LIN {X 0,Y 523.259,Z 482.213,A -85,B 0,C 180,E1 -4769.999,E2 -4769.999} C_VEL
LIN {X 0,Y 523.274,Z 481.391,A -85,B 0,C 180,E1 -4771.538,E2 -4771.538} C_VEL
LIN {X 0,Y 523.335,Z 480.397,A -85,B 0,C 180,E1 -4772.307,E2 -4772.307} C_VEL
LIN {X 0,Y 523.367,Z 478.999,A -85,B 0,C 180,E1 -4773.077,E2 -4773.077} C_VEL
LIN {X 0,Y 523.423,Z 476.057,A -85,B 0,C 180,E1 -4774.233,E2 -4774.233} C_VEL
LIN {X 0,Y 523.455,Z 472.072,A -85,B 0,C 180,E1 -4775.391,E2 -4775.391} C_VEL
LIN {X 0,Y 523.508,Z 466.867,A -85,B 0,C 180,E1 -4776.566,E2 -4776.566} C_VEL
LIN {X 0,Y 523.611,Z 460.488,A -85,B 0,C 180,E1 -4777.711,E2 -4777.711} C_VEL
LIN {X 0,Y 523.8,Z 452.437,A -85,B 0,C 180,E1 -4778.874,E2 -4778.874} C_VEL
LIN {X 0,Y 523.986,Z 444.235,A -85,B 0,C 180,E1 -4779.844,E2 -4779.844} C_VEL
LIN {X 0,Y 524.294,Z 434.24,A -85,B 0,C 180,E1 -4780.814,E2 -4780.814} C_VEL
LIN {X 0,Y 524.558,Z 422.98,A -85,B 0,C 180,E1 -4781.687,E2 -4781.687} C_VEL
LIN {X 0,Y 524.835,Z 411.905,A -85,B 0,C 180,E1 -4782.369,E2 -4782.369} C_VEL
LIN {X 0,Y 525.111,Z 399.665,A -85,B 0,C 180,E1 -4782.952,E2 -4782.952} C_VEL
LIN {X 0,Y 525.344,Z 387.753,A -85,B 0,C 180,E1 -4783.364,E2 -4783.364} C_VEL
LIN {X 0,Y 525.517,Z 374.759,A -85,B 0,C 180,E1 -4783.655,E2 -4783.655} C_VEL
LIN {X 0,Y 525.809,Z 279.444,A -85,B 0,C 180,E1 -4784.972,E2 -4784.972} C_VEL
LIN {X 0,Y 524.262,Z 268.901,A -85,B 0,C 180,E1 -4785.178,E2 -4785.178} C_VEL
LIN {X 0,Y 524.642,Z 248.982,A -85,B 0,C 180,E1 -4788.123,E2 -4788.123} C_VEL
LIN {X 0,Y 525.091,Z 228.582,A -85,B 0,C 180,E1 -4791.181,E2 -4791.181} C_VEL
LIN {X 0,Y 525.423,Z 212.316,A -85,B 0,C 180,E1 -4793.654,E2 -4793.654} C_VEL
LIN {X 0,Y 523.985,Z 204.216,A -85,B 0,C 180,E1 -4794.988,E2 -4794.988} C_VEL
LIN {X 0,Y 523.955,Z 204.222,A -85,B 0,C 180,E1 -4797.995,E2 -4797.995} C_VEL
LIN {X 0,Y 523.926,Z 204.218,A -85,B 0,C 180,E1 -4800.851,E2 -4800.851} C_VEL
LIN {X 0,Y 523.942,Z 204.22,A -85,B 0,C 180,E1 -4803.731,E2 -4803.731} C_VEL
LIN {X 0,Y 523.898,Z 204.224,A -85,B 0,C 180,E1 -4806.4,E2 -4806.4} C_VEL
LIN {X 0,Y 523.896,Z 204.221,A -85,B 0,C 180,E1 -4809.08,E2 -4809.08} C_VEL
LIN {X 0,Y 523.926,Z 204.223,A -85,B 0,C 180,E1 -4812.114,E2 -4812.114} C_VEL
LIN {X 0,Y 523.922,Z 204.22,A -85,B 0,C 180,E1 -4815.305,E2 -4815.305} C_VEL
LIN {X 0,Y 523.946,Z 204.215,A -85,B 0,C 180,E1 -4818.682,E2 -4818.682} C_VEL
LIN {X 0,Y 523.916,Z 204.22,A -85,B 0,C 180,E1 -4821.072,E2 -4821.072} C_VEL
LIN {X 0,Y 523.887,Z 204.229,A -85,B 0,C 180,E1 -4823.824,E2 -4823.824} C_VEL
LIN {X 0,Y 523.904,Z 204.22,A -85,B 0,C 180,E1 -4826.633,E2 -4826.633} C_VEL
LIN {X 0,Y 523.918,Z 204.224,A -85,B 0,C 180,E1 -4829.353,E2 -4829.353} C_VEL
LIN {X 0,Y 523.932,Z 204.217,A -85,B 0,C 180,E1 -4832.277,E2 -4832.277} C_VEL
LIN {X 0,Y 523.904,Z 204.22,A -85,B 0,C 180,E1 -4834.579,E2 -4834.579} C_VEL
LIN {X 0,Y 523.913,Z 204.223,A -85,B 0,C 180,E1 -4837.107,E2 -4837.107} C_VEL
LIN {X 0,Y 523.925,Z 204.22,A -85,B 0,C 180,E1 -4839.863,E2 -4839.863} C_VEL
LIN {X 0,Y 523.941,Z 204.218,A -85,B 0,C 180,E1 -4842.836,E2 -4842.836} C_VEL
LIN {X 0,Y 523.945,Z 204.223,A -85,B 0,C 180,E1 -4845.235,E2 -4845.235} C_VEL
LIN {X 0,Y 523.959,Z 204.213,A -85,B 0,C 180,E1 -4848.393,E2 -4848.393} C_VEL
LIN {X 0,Y 523.95,Z 204.219,A -85,B 0,C 180,E1 -4851.515,E2 -4851.515} C_VEL
LIN {X 0,Y 523.993,Z 204.21,A -85,B 0,C 180,E1 -4853.84,E2 -4853.84} C_VEL
LIN {X 0,Y 524.021,Z 204.212,A -85,B 0,C 180,E1 -4856.925,E2 -4856.925} C_VEL
LIN {X 0,Y 524.047,Z 204.202,A -85,B 0,C 180,E1 -4860,E2 -4860} C_VEL
LIN {X 0,Y 524.019,Z 204.214,A -85,B 0,C 180,E1 -4863.075,E2 -4863.075} C_VEL
LIN {X 0,Y 523.985,Z 204.21,A -85,B 0,C 180,E1 -4866.16,E2 -4866.16} C_VEL
LIN {X 0,Y 523.948,Z 204.218,A -85,B 0,C 180,E1 -4869.263,E2 -4869.263} C_VEL
LIN {X 0,Y 523.965,Z 204.212,A -85,B 0,C 180,E1 -4871.753,E2 -4871.753} C_VEL
LIN {X 0,Y 523.934,Z 204.221,A -85,B 0,C 180,E1 -4875.054,E2 -4875.054} C_VEL
LIN {X 0,Y 523.915,Z 204.219,A -85,B 0,C 180,E1 -4877.971,E2 -4877.971} C_VEL
LIN {X 0,Y 523.918,Z 204.223,A -85,B 0,C 180,E1 -4880.412,E2 -4880.412} C_VEL
LIN {X 0,Y 523.89,Z 204.227,A -85,B 0,C 180,E1 -4882.895,E2 -4882.895} C_VEL
LIN {X 0,Y 523.934,Z 204.218,A -85,B 0,C 180,E1 -4886.023,E2 -4886.023} C_VEL
LIN {X 0,Y 523.911,Z 204.223,A -85,B 0,C 180,E1 -4888.877,E2 -4888.877} C_VEL
LIN {X 0,Y 523.886,Z 204.222,A -85,B 0,C 180,E1 -4891.547,E2 -4891.547} C_VEL
LIN {X 0,Y 523.902,Z 204.227,A -85,B 0,C 180,E1 -4894.293,E2 -4894.293} C_VEL
LIN {X 0,Y 523.871,Z 204.225,A -85,B 0,C 180,E1 -4897.135,E2 -4897.135} C_VEL
LIN {X 0,Y 523.931,Z 204.223,A -85,B 0,C 180,E1 -4900.138,E2 -4900.138} C_VEL
LIN {X 0,Y 523.89,Z 204.222,A -85,B 0,C 180,E1 -4903.17,E2 -4903.17} C_VEL
LIN {X 0,Y 523.907,Z 204.222,A -85,B 0,C 180,E1 -4905.776,E2 -4905.776} C_VEL
LIN {X 0,Y 523.887,Z 204.223,A -85,B 0,C 180,E1 -4906.947,E2 -4906.947} C_VEL
LIN {X 0,Y 523.224,Z 204.307,A -85,B 0,C 180,E1 -4907.589,E2 -4907.589} C_VEL
LIN {X 0,Y 520.381,Z 204.668,A -85,B 0,C 180,E1 -4908.631,E2 -4908.631} C_VEL
LIN {X 0,Y 517.975,Z 204.971,A -85,B 0,C 180,E1 -4909.47,E2 -4909.47} C_VEL
LIN {X 0,Y 516.94,Z 205.097,A -85,B 0,C 180,E1 -4910.118,E2 -4910.118} C_VEL
LIN {X 0,Y 516.854,Z 205.105,A -85,B 0,C 180,E1 -4910.337,E2 -4910.337} C_VEL
LIN {X 0,Y 516.861,Z 205.098,A -85,B 0,C 180,E1 -4913.346,E2 -4913.346} C_VEL
LIN {X 0,Y 516.89,Z 205.102,A -85,B 0,C 180,E1 -4916.125,E2 -4916.125} C_VEL
LIN {X 0,Y 516.874,Z 205.096,A -85,B 0,C 180,E1 -4918.94,E2 -4918.94} C_VEL
LIN {X 0,Y 516.903,Z 205.096,A -85,B 0,C 180,E1 -4921.589,E2 -4921.589} C_VEL
LIN {X 0,Y 516.917,Z 205.095,A -85,B 0,C 180,E1 -4924.214,E2 -4924.214} C_VEL
LIN {X 0,Y 516.85,Z 205.099,A -85,B 0,C 180,E1 -4926.78,E2 -4926.78} C_VEL
LIN {X 0,Y 516.932,Z 205.096,A -85,B 0,C 180,E1 -4929.735,E2 -4929.735} C_VEL
LIN {X 0,Y 516.889,Z 205.094,A -85,B 0,C 180,E1 -4932.598,E2 -4932.598} C_VEL
LIN {X 0,Y 516.932,Z 205.089,A -85,B 0,C 180,E1 -4935.033,E2 -4935.033} C_VEL
LIN {X 0,Y 516.965,Z 205.089,A -85,B 0,C 180,E1 -4938.236,E2 -4938.236} C_VEL
LIN {X 0,Y 516.992,Z 205.09,A -85,B 0,C 180,E1 -4941.796,E2 -4941.796} C_VEL
LIN {X 0,Y 517.024,Z 205.25,A -85,B 0,C 180,E1 -4942.042,E2 -4942.042} C_VEL
LIN {X 0,Y 517.431,Z 211.036,A -85,B 0,C 180,E1 -4943.177,E2 -4943.177} C_VEL
LIN {X 0,Y 517.244,Z 221.184,A -85,B 0,C 180,E1 -4945.13,E2 -4945.13} C_VEL
LIN {X 0,Y 517.148,Z 224.133,A -85,B 0,C 180,E1 -4945.691,E2 -4945.691} C_VEL
LIN {X 0,Y 519.152,Z 234.665,A -85,B 0,C 180,E1 -4945.902,E2 -4945.902} C_VEL
LIN {X 0,Y 518.617,Z 330.957,A -85,B 0,C 180,E1 -4947.259,E2 -4947.259} C_VEL
LIN {X 0,Y 518.459,Z 344.692,A -85,B 0,C 180,E1 -4947.622,E2 -4947.622} C_VEL
LIN {X 0,Y 518.225,Z 357.03,A -85,B 0,C 180,E1 -4948.107,E2 -4948.107} C_VEL
LIN {X 0,Y 517.963,Z 368.835,A -85,B 0,C 180,E1 -4948.738,E2 -4948.738} C_VEL
LIN {X 0,Y 517.567,Z 380.167,A -85,B 0,C 180,E1 -4949.515,E2 -4949.515} C_VEL
LIN {X 0,Y 517.288,Z 390.365,A -85,B 0,C 180,E1 -4950.391,E2 -4950.391} C_VEL
LIN {X 0,Y 517.054,Z 399.569,A -85,B 0,C 180,E1 -4951.364,E2 -4951.364} C_VEL
LIN {X 0,Y 516.777,Z 408.492,A -85,B 0,C 180,E1 -4952.534,E2 -4952.534} C_VEL
LIN {X 0,Y 516.608,Z 415.7,A -85,B 0,C 180,E1 -4953.706,E2 -4953.706} C_VEL
LIN {X 0,Y 516.537,Z 420.592,A -85,B 0,C 180,E1 -4954.684,E2 -4954.684} C_VEL
LIN {X 0,Y 516.428,Z 425.363,A -85,B 0,C 180,E1 -4955.859,E2 -4955.859} C_VEL
LIN {X 0,Y 516.346,Z 429.038,A -85,B 0,C 180,E1 -4957.037,E2 -4957.037} C_VEL
LIN {X 0,Y 516.302,Z 430.941,A -85,B 0,C 180,E1 -4957.824,E2 -4957.824} C_VEL
LIN {X 0,Y 516.256,Z 432.404,A -85,B 0,C 180,E1 -4958.613,E2 -4958.613} C_VEL
LIN {X 0,Y 516.253,Z 434.068,A -85,B 0,C 180,E1 -4960.194,E2 -4960.194} C_VEL
LIN {X 0,Y 516.285,Z 434.25,A -85,B 0,C 180,E1 -4961.445,E2 -4961.445} C_VEL
LIN {X 0,Y 516.225,Z 433.544,A -85,B 0,C 180,E1 -4962.582,E2 -4962.582} C_VEL
LIN {X 0,Y 516.226,Z 432.549,A -85,B 0,C 180,E1 -4963.382,E2 -4963.382} C_VEL
LIN {X 0,Y 516.284,Z 431.135,A -85,B 0,C 180,E1 -4964.184,E2 -4964.184} C_VEL
LIN {X 0,Y 516.358,Z 428.136,A -85,B 0,C 180,E1 -4965.391,E2 -4965.391} C_VEL
LIN {X 0,Y 516.417,Z 424.022,A -85,B 0,C 180,E1 -4966.606,E2 -4966.606} C_VEL
LIN {X 0,Y 516.585,Z 418.042,A -85,B 0,C 180,E1 -4967.943,E2 -4967.943} C_VEL
LIN {X 0,Y 516.752,Z 410.539,A -85,B 0,C 180,E1 -4969.257,E2 -4969.257} C_VEL
LIN {X 0,Y 517.011,Z 401.987,A -85,B 0,C 180,E1 -4970.436,E2 -4970.436} C_VEL
LIN {X 0,Y 517.31,Z 392.237,A -85,B 0,C 180,E1 -4971.519,E2 -4971.519} C_VEL
LIN {X 0,Y 517.56,Z 383.089,A -85,B 0,C 180,E1 -4972.346,E2 -4972.346} C_VEL
LIN {X 0,Y 517.908,Z 371.737,A -85,B 0,C 180,E1 -4973.173,E2 -4973.173} C_VEL
LIN {X 0,Y 518.157,Z 359.819,A -85,B 0,C 180,E1 -4973.85,E2 -4973.85} C_VEL
LIN {X 0,Y 518.398,Z 346.983,A -85,B 0,C 180,E1 -4974.395,E2 -4974.395} C_VEL
LIN {X 0,Y 518.591,Z 333.832,A -85,B 0,C 180,E1 -4974.77,E2 -4974.77} C_VEL
LIN {X 0,Y 518.727,Z 314.797,A -85,B 0,C 180,E1 -4975.075,E2 -4975.075} C_VEL
LIN {X 0,Y 519.05,Z 233.791,A -85,B 0,C 180,E1 -4976.205,E2 -4976.205} C_VEL
LIN {X 0,Y 517.227,Z 224.102,A -85,B 0,C 180,E1 -4976.404,E2 -4976.404} C_VEL
LIN {X 0,Y 517.324,Z 208.898,A -85,B 0,C 180,E1 -4979.278,E2 -4979.278} C_VEL
LIN {X 0,Y 516.97,Z 205.092,A -85,B 0,C 180,E1 -4980.027,E2 -4980.027} C_VEL
LIN {X 0,Y 516.891,Z 205.098,A -85,B 0,C 180,E1 -4982.945,E2 -4982.945} C_VEL
LIN {X 0,Y 516.885,Z 205.098,A -85,B 0,C 180,E1 -4985.777,E2 -4985.777} C_VEL
LIN {X 0,Y 516.877,Z 205.102,A -85,B 0,C 180,E1 -4988.714,E2 -4988.714} C_VEL
LIN {X 0,Y 516.907,Z 205.097,A -85,B 0,C 180,E1 -4991.773,E2 -4991.773} C_VEL
LIN {X 0,Y 516.909,Z 205.093,A -85,B 0,C 180,E1 -4995.008,E2 -4995.008} C_VEL
LIN {X 0,Y 516.907,Z 205.098,A -85,B 0,C 180,E1 -4998.396,E2 -4998.396} C_VEL
LIN {X 0,Y 516.867,Z 205.098,A -85,B 0,C 180,E1 -5001.283,E2 -5001.283} C_VEL
LIN {X 0,Y 516.87,Z 205.102,A -85,B 0,C 180,E1 -5004.219,E2 -5004.219} C_VEL
LIN {X 0,Y 516.876,Z 205.096,A -85,B 0,C 180,E1 -5007.051,E2 -5007.051} C_VEL
LIN {X 0,Y 516.877,Z 205.102,A -85,B 0,C 180,E1 -5009.795,E2 -5009.795} C_VEL
LIN {X 0,Y 516.904,Z 205.091,A -85,B 0,C 180,E1 -5012.466,E2 -5012.466} C_VEL
LIN {X 0,Y 516.886,Z 205.096,A -85,B 0,C 180,E1 -5015.07,E2 -5015.07} C_VEL
LIN {X 0,Y 516.884,Z 205.101,A -85,B 0,C 180,E1 -5017.622,E2 -5017.622} C_VEL
LIN {X 0,Y 516.902,Z 205.093,A -85,B 0,C 180,E1 -5020.128,E2 -5020.128} C_VEL
LIN {X 0,Y 516.911,Z 205.092,A -85,B 0,C 180,E1 -5022.595,E2 -5022.595} C_VEL
LIN {X 0,Y 516.908,Z 205.092,A -85,B 0,C 180,E1 -5025.029,E2 -5025.029} C_VEL
LIN {X 0,Y 516.932,Z 205.088,A -85,B 0,C 180,E1 -5028.233,E2 -5028.233} C_VEL
LIN {X 0,Y 516.938,Z 205.097,A -85,B 0,C 180,E1 -5031.399,E2 -5031.399} C_VEL
LIN {X 0,Y 516.983,Z 205.084,A -85,B 0,C 180,E1 -5033.756,E2 -5033.756} C_VEL
LIN {X 0,Y 516.981,Z 205.086,A -85,B 0,C 180,E1 -5036.883,E2 -5036.883} C_VEL
LIN {X 0,Y 517.042,Z 205.076,A -85,B 0,C 180,E1 -5040,E2 -5040} C_VEL
LIN {X 0,Y 516.98,Z 205.088,A -85,B 0,C 180,E1 -5043.117,E2 -5043.117} C_VEL
LIN {X 0,Y 516.964,Z 205.085,A -85,B 0,C 180,E1 -5046.244,E2 -5046.244} C_VEL
LIN {X 0,Y 516.918,Z 205.094,A -85,B 0,C 180,E1 -5049.39,E2 -5049.39} C_VEL
LIN {X 0,Y 516.95,Z 205.085,A -85,B 0,C 180,E1 -5051.825,E2 -5051.825} C_VEL
LIN {X 0,Y 516.909,Z 205.096,A -85,B 0,C 180,E1 -5055.147,E2 -5055.147} C_VEL
LIN {X 0,Y 516.882,Z 205.095,A -85,B 0,C 180,E1 -5058.224,E2 -5058.224} C_VEL
LIN {X 0,Y 516.88,Z 205.102,A -85,B 0,C 180,E1 -5060.703,E2 -5060.703} C_VEL
LIN {X 0,Y 516.857,Z 205.1,A -85,B 0,C 180,E1 -5064.075,E2 -5064.075} C_VEL
LIN {X 0,Y 516.868,Z 205.104,A -85,B 0,C 180,E1 -5066.661,E2 -5066.661} C_VEL
LIN {X 0,Y 516.881,Z 205.093,A -85,B 0,C 180,E1 -5069.525,E2 -5069.525} C_VEL
LIN {X 0,Y 516.868,Z 205.103,A -85,B 0,C 180,E1 -5072.545,E2 -5072.545} C_VEL
LIN {X 0,Y 516.841,Z 205.101,A -85,B 0,C 180,E1 -5075.331,E2 -5075.331} C_VEL
LIN {X 0,Y 516.857,Z 205.097,A -85,B 0,C 180,E1 -5077.944,E2 -5077.944} C_VEL
LIN {X 0,Y 516.865,Z 205.101,A -85,B 0,C 180,E1 -5080.744,E2 -5080.744} C_VEL
LIN {X 0,Y 516.865,Z 205.099,A -85,B 0,C 180,E1 -5082.833,E2 -5082.833} C_VEL
LIN {X 0,Y 516.88,Z 205.095,A -85,B 0,C 180,E1 -5085.009,E2 -5085.009} C_VEL
LIN {X 0,Y 516.889,Z 205.099,A -85,B 0,C 180,E1 -5088.402,E2 -5088.402} C_VEL
LIN {X 0,Y 516.866,Z 205.097,A -85,B 0,C 180,E1 -5091.285,E2 -5091.285} C_VEL
LIN {X 0,Y 516.866,Z 205.102,A -85,B 0,C 180,E1 -5094.222,E2 -5094.222} C_VEL
LIN {X 0,Y 516.888,Z 205.094,A -85,B 0,C 180,E1 -5097.054,E2 -5097.054} C_VEL
LIN {X 0,Y 516.887,Z 205.103,A -85,B 0,C 180,E1 -5099.798,E2 -5099.798} C_VEL
LIN {X 0,Y 516.894,Z 205.098,A -85,B 0,C 180,E1 -5102.467,E2 -5102.467} C_VEL
LIN {X 0,Y 516.938,Z 205.256,A -85,B 0,C 180,E1 -5104.913,E2 -5104.913} C_VEL
LIN {X 0,Y 518.407,Z 213.106,A -85,B 0,C 180,E1 -5106.215,E2 -5106.215} C_VEL
LIN {X 0,Y 518.263,Z 223.955,A -85,B 0,C 180,E1 -5107.895,E2 -5107.895} C_VEL
LIN {X 0,Y 517.773,Z 242.933,A -85,B 0,C 180,E1 -5110.783,E2 -5110.783} C_VEL
LIN {X 0,Y 517.374,Z 261.888,A -85,B 0,C 180,E1 -5113.628,E2 -5113.628} C_VEL
LIN {X 0,Y 517.226,Z 268.541,A -85,B 0,C 180,E1 -5114.62,E2 -5114.62} C_VEL
LIN {X 0,Y 519.036,Z 280.742,A -85,B 0,C 180,E1 -5114.852,E2 -5114.852} C_VEL
LIN {X 0,Y 518.608,Z 377.04,A -85,B 0,C 180,E1 -5116.206,E2 -5116.206} C_VEL
LIN {X 0,Y 518.342,Z 390.389,A -85,B 0,C 180,E1 -5116.549,E2 -5116.549} C_VEL
LIN {X 0,Y 518.022,Z 403.73,A -85,B 0,C 180,E1 -5117.064,E2 -5117.064} C_VEL
LIN {X 0,Y 517.792,Z 415.956,A -85,B 0,C 180,E1 -5117.72,E2 -5117.72} C_VEL
LIN {X 0,Y 517.447,Z 427.872,A -85,B 0,C 180,E1 -5118.542,E2 -5118.542} C_VEL
LIN {X 0,Y 517.149,Z 438.108,A -85,B 0,C 180,E1 -5119.428,E2 -5119.428} C_VEL
LIN {X 0,Y 516.872,Z 447.319,A -85,B 0,C 180,E1 -5120.411,E2 -5120.411} C_VEL
LIN {X 0,Y 516.655,Z 456.298,A -85,B 0,C 180,E1 -5121.591,E2 -5121.591} C_VEL
LIN {X 0,Y 516.503,Z 463.529,A -85,B 0,C 180,E1 -5122.769,E2 -5122.769} C_VEL
LIN {X 0,Y 516.402,Z 470.115,A -85,B 0,C 180,E1 -5124.141,E2 -5124.141} C_VEL
LIN {X 0,Y 516.268,Z 474.471,A -85,B 0,C 180,E1 -5125.314,E2 -5125.314} C_VEL
LIN {X 0,Y 516.352,Z 476.783,A -85,B 0,C 180,E1 -5126.097,E2 -5126.097} C_VEL
LIN {X 0,Y 516.283,Z 478.653,A -85,B 0,C 180,E1 -5126.877,E2 -5126.877} C_VEL
LIN {X 0,Y 516.261,Z 480.056,A -85,B 0,C 180,E1 -5127.658,E2 -5127.658} C_VEL
LIN {X 0,Y 516.167,Z 481.667,A -85,B 0,C 180,E1 -5129.218,E2 -5129.218} C_VEL
LIN {X 0,Y 516.167,Z 481.887,A -85,B 0,C 180,E1 -5129.999,E2 -5129.999} C_VEL
LIN {X 0,Y 516.192,Z 481.066,A -85,B 0,C 180,E1 -5131.559,E2 -5131.559} C_VEL
LIN {X 0,Y 516.261,Z 480.072,A -85,B 0,C 180,E1 -5132.339,E2 -5132.339} C_VEL
LIN {X 0,Y 516.282,Z 478.673,A -85,B 0,C 180,E1 -5133.12,E2 -5133.12} C_VEL
LIN {X 0,Y 516.311,Z 475.73,A -85,B 0,C 180,E1 -5134.292,E2 -5134.292} C_VEL
LIN {X 0,Y 516.368,Z 471.746,A -85,B 0,C 180,E1 -5135.465,E2 -5135.465} C_VEL
LIN {X 0,Y 516.442,Z 465.838,A -85,B 0,C 180,E1 -5136.794,E2 -5136.794} C_VEL
LIN {X 0,Y 516.59,Z 458.92,A -85,B 0,C 180,E1 -5138.014,E2 -5138.014} C_VEL
LIN {X 0,Y 516.772,Z 450.612,A -85,B 0,C 180,E1 -5139.193,E2 -5139.193} C_VEL
LIN {X 0,Y 516.997,Z 442.1,A -85,B 0,C 180,E1 -5140.176,E2 -5140.176} C_VEL
LIN {X 0,Y 517.333,Z 431.588,A -85,B 0,C 180,E1 -5141.16,E2 -5141.16} C_VEL
LIN {X 0,Y 517.673,Z 420.381,A -85,B 0,C 180,E1 -5142.002,E2 -5142.002} C_VEL
LIN {X 0,Y 517.924,Z 409.797,A -85,B 0,C 180,E1 -5142.636,E2 -5142.636} C_VEL
LIN {X 0,Y 518.19,Z 398.114,A -85,B 0,C 180,E1 -5143.178,E2 -5143.178} C_VEL
LIN {X 0,Y 518.448,Z 385.577,A -85,B 0,C 180,E1 -5143.595,E2 -5143.595} C_VEL
LIN {X 0,Y 518.644,Z 372.898,A -85,B 0,C 180,E1 -5143.865,E2 -5143.865} C_VEL
LIN {X 0,Y 518.944,Z 280.255,A -85,B 0,C 180,E1 -5145.159,E2 -5145.159} C_VEL
LIN {X 0,Y 517.245,Z 268.532,A -85,B 0,C 180,E1 -5145.394,E2 -5145.394} C_VEL
LIN {X 0,Y 517.686,Z 248.534,A -85,B 0,C 180,E1 -5148.396,E2 -5148.396} C_VEL
LIN {X 0,Y 518.169,Z 228.255,A -85,B 0,C 180,E1 -5151.478,E2 -5151.478} C_VEL
LIN {X 0,Y 518.543,Z 214.679,A -85,B 0,C 180,E1 -5153.563,E2 -5153.563} C_VEL
LIN {X 0,Y 517.179,Z 206.415,A -85,B 0,C 180,E1 -5154.91,E2 -5154.91} C_VEL
LIN {X 0,Y 516.93,Z 205.095,A -85,B 0,C 180,E1 -5155.138,E2 -5155.138} C_VEL
LIN {X 0,Y 516.912,Z 205.099,A -85,B 0,C 180,E1 -5157.902,E2 -5157.902} C_VEL
LIN {X 0,Y 516.875,Z 205.103,A -85,B 0,C 180,E1 -5160.2,E2 -5160.2} C_VEL
LIN {X 0,Y 516.877,Z 205.095,A -85,B 0,C 180,E1 -5162.943,E2 -5162.943} C_VEL
LIN {X 0,Y 516.868,Z 205.102,A -85,B 0,C 180,E1 -5165.775,E2 -5165.775} C_VEL
LIN {X 0,Y 516.856,Z 205.098,A -85,B 0,C 180,E1 -5168.712,E2 -5168.712} C_VEL
LIN {X 0,Y 516.886,Z 205.102,A -85,B 0,C 180,E1 -5171.771,E2 -5171.771} C_VEL
LIN {X 0,Y 516.89,Z 205.094,A -85,B 0,C 180,E1 -5175.006,E2 -5175.006} C_VEL
LIN {X 0,Y 516.893,Z 205.095,A -85,B 0,C 180,E1 -5178.393,E2 -5178.393} C_VEL
LIN {X 0,Y 516.868,Z 205.099,A -85,B 0,C 180,E1 -5181.283,E2 -5181.283} C_VEL
LIN {X 0,Y 516.849,Z 205.101,A -85,B 0,C 180,E1 -5184.218,E2 -5184.218} C_VEL
LIN {X 0,Y 516.86,Z 205.099,A -85,B 0,C 180,E1 -5187.05,E2 -5187.05} C_VEL
LIN {X 0,Y 516.857,Z 205.104,A -85,B 0,C 180,E1 -5189.794,E2 -5189.794} C_VEL
LIN {X 0,Y 516.881,Z 205.095,A -85,B 0,C 180,E1 -5192.465,E2 -5192.465} C_VEL
LIN {X 0,Y 516.871,Z 205.099,A -85,B 0,C 180,E1 -5195.07,E2 -5195.07} C_VEL
LIN {X 0,Y 516.878,Z 205.102,A -85,B 0,C 180,E1 -5197.622,E2 -5197.622} C_VEL
LIN {X 0,Y 516.878,Z 205.096,A -85,B 0,C 180,E1 -5200.128,E2 -5200.128} C_VEL
LIN {X 0,Y 516.886,Z 205.095,A -85,B 0,C 180,E1 -5202.595,E2 -5202.595} C_VEL
LIN {X 0,Y 516.852,Z 205.1,A -85,B 0,C 180,E1 -5205.832,E2 -5205.832} C_VEL
LIN {X 0,Y 516.945,Z 205.087,A -85,B 0,C 180,E1 -5208.233,E2 -5208.233} C_VEL
LIN {X 0,Y 516.915,Z 205.097,A -85,B 0,C 180,E1 -5211.399,E2 -5211.399} C_VEL
LIN {X 0,Y 516.961,Z 205.086,A -85,B 0,C 180,E1 -5213.756,E2 -5213.756} C_VEL
LIN {X 0,Y 516.987,Z 205.088,A -85,B 0,C 180,E1 -5216.883,E2 -5216.883} C_VEL
LIN {X 0,Y 517.018,Z 205.078,A -85,B 0,C 180,E1 -5220,E2 -5220} C_VEL
LIN {X 0,Y 516.959,Z 205.092,A -85,B 0,C 180,E1 -5223.117,E2 -5223.117} C_VEL
LIN {X 0,Y 516.949,Z 205.087,A -85,B 0,C 180,E1 -5226.244,E2 -5226.244} C_VEL
LIN {X 0,Y 516.903,Z 205.094,A -85,B 0,C 180,E1 -5229.39,E2 -5229.39} C_VEL
LIN {X 0,Y 516.924,Z 205.089,A -85,B 0,C 180,E1 -5231.826,E2 -5231.826} C_VEL
LIN {X 0,Y 516.888,Z 205.098,A -85,B 0,C 180,E1 -5235.149,E2 -5235.149} C_VEL
LIN {X 0,Y 516.874,Z 205.098,A -85,B 0,C 180,E1 -5238.224,E2 -5238.224} C_VEL
LIN {X 0,Y 516.861,Z 205.106,A -85,B 0,C 180,E1 -5240.704,E2 -5240.704} C_VEL
LIN {X 0,Y 516.838,Z 205.102,A -85,B 0,C 180,E1 -5243.225,E2 -5243.225} C_VEL
LIN {X 0,Y 516.893,Z 205.097,A -85,B 0,C 180,E1 -5246.199,E2 -5246.199} C_VEL
LIN {X 0,Y 516.895,Z 205.094,A -85,B 0,C 180,E1 -5249.306,E2 -5249.306} C_VEL
LIN {X 0,Y 516.856,Z 205.106,A -85,B 0,C 180,E1 -5252.548,E2 -5252.548} C_VEL
LIN {X 0,Y 516.841,Z 205.1,A -85,B 0,C 180,E1 -5255.336,E2 -5255.336} C_VEL
LIN {X 0,Y 516.841,Z 205.103,A -85,B 0,C 180,E1 -5257.947,E2 -5257.947} C_VEL
LIN {X 0,Y 516.867,Z 205.1,A -85,B 0,C 180,E1 -5260.744,E2 -5260.744} C_VEL
LIN {X 0,Y 516.849,Z 205.103,A -85,B 0,C 180,E1 -5263.907,E2 -5263.907} C_VEL
LIN {X 0,Y 516.851,Z 205.106,A -85,B 0,C 180,E1 -5266.111,E2 -5266.111} C_VEL
LIN {X 0,Y 516.888,Z 205.1,A -85,B 0,C 180,E1 -5268.402,E2 -5268.402} C_VEL
LIN {X 0,Y 516.854,Z 205.105,A -85,B 0,C 180,E1 -5270.337,E2 -5270.337} C_VEL
LIN {X 0,Y 516.186,Z 205.184,A -85,B 0,C 180,E1 -5270.987,E2 -5270.987} C_VEL
LIN {X 0,Y 513.34,Z 205.544,A -85,B 0,C 180,E1 -5272.043,E2 -5272.043} C_VEL
LIN {X 0,Y 510.933,Z 205.842,A -85,B 0,C 180,E1 -5272.894,E2 -5272.894} C_VEL
LIN {X 0,Y 509.894,Z 205.968,A -85,B 0,C 180,E1 -5273.551,E2 -5273.551} C_VEL
LIN {X 0,Y 509.806,Z 205.978,A -85,B 0,C 180,E1 -5273.773,E2 -5273.773} C_VEL
LIN {X 0,Y 509.841,Z 205.974,A -85,B 0,C 180,E1 -5276.543,E2 -5276.543} C_VEL
LIN {X 0,Y 509.829,Z 205.974,A -85,B 0,C 180,E1 -5279.338,E2 -5279.338} C_VEL
LIN {X 0,Y 509.877,Z 205.975,A -85,B 0,C 180,E1 -5282.058,E2 -5282.058} C_VEL
LIN {X 0,Y 509.828,Z 205.974,A -85,B 0,C 180,E1 -5284.706,E2 -5284.706} C_VEL
LIN {X 0,Y 509.817,Z 205.978,A -85,B 0,C 180,E1 -5287.462,E2 -5287.462} C_VEL
LIN {X 0,Y 509.909,Z 205.972,A -85,B 0,C 180,E1 -5289.848,E2 -5289.848} C_VEL
LIN {X 0,Y 509.857,Z 205.971,A -85,B 0,C 180,E1 -5293.177,E2 -5293.177} C_VEL
LIN {X 0,Y 509.851,Z 205.978,A -85,B 0,C 180,E1 -5295.637,E2 -5295.637} C_VEL
LIN {X 0,Y 509.911,Z 205.966,A -85,B 0,C 180,E1 -5298.877,E2 -5298.877} C_VEL
LIN {X 0,Y 509.972,Z 206.155,A -85,B 0,C 180,E1 -5301.932,E2 -5301.932} C_VEL
LIN {X 0,Y 510.451,Z 211.978,A -85,B 0,C 180,E1 -5303.083,E2 -5303.083} C_VEL
LIN {X 0,Y 510.249,Z 222.23,A -85,B 0,C 180,E1 -5305.064,E2 -5305.064} C_VEL
LIN {X 0,Y 510.173,Z 224.48,A -85,B 0,C 180,E1 -5305.477,E2 -5305.477} C_VEL
LIN {X 0,Y 512.314,Z 235.3,A -85,B 0,C 180,E1 -5305.699,E2 -5305.699} C_VEL
LIN {X 0,Y 511.729,Z 331.459,A -85,B 0,C 180,E1 -5307.074,E2 -5307.074} C_VEL
LIN {X 0,Y 511.56,Z 345.133,A -85,B 0,C 180,E1 -5307.443,E2 -5307.443} C_VEL
LIN {X 0,Y 511.317,Z 357.436,A -85,B 0,C 180,E1 -5307.934,E2 -5307.934} C_VEL
LIN {X 0,Y 511.073,Z 368.435,A -85,B 0,C 180,E1 -5308.524,E2 -5308.524} C_VEL
LIN {X 0,Y 510.64,Z 379.904,A -85,B 0,C 180,E1 -5309.312,E2 -5309.312} C_VEL
LIN {X 0,Y 510.345,Z 390.2,A -85,B 0,C 180,E1 -5310.199,E2 -5310.199} C_VEL
LIN {X 0,Y 510.096,Z 399.507,A -85,B 0,C 180,E1 -5311.186,E2 -5311.186} C_VEL
LIN {X 0,Y 509.752,Z 408.512,A -85,B 0,C 180,E1 -5312.372,E2 -5312.372} C_VEL
LIN {X 0,Y 509.563,Z 415.773,A -85,B 0,C 180,E1 -5313.559,E2 -5313.559} C_VEL
LIN {X 0,Y 509.473,Z 421.607,A -85,B 0,C 180,E1 -5314.749,E2 -5314.749} C_VEL
LIN {X 0,Y 509.364,Z 426.233,A -85,B 0,C 180,E1 -5315.941,E2 -5315.941} C_VEL
LIN {X 0,Y 509.273,Z 429.773,A -85,B 0,C 180,E1 -5317.135,E2 -5317.135} C_VEL
LIN {X 0,Y 509.202,Z 431.588,A -85,B 0,C 180,E1 -5317.934,E2 -5317.934} C_VEL
LIN {X 0,Y 509.157,Z 432.947,A -85,B 0,C 180,E1 -5318.734,E2 -5318.734} C_VEL
LIN {X 0,Y 509.188,Z 434.487,A -85,B 0,C 180,E1 -5320.337,E2 -5320.337} C_VEL
LIN {X 0,Y 509.188,Z 434.571,A -85,B 0,C 180,E1 -5321.486,E2 -5321.486} C_VEL
LIN {X 0,Y 509.144,Z 433.715,A -85,B 0,C 180,E1 -5322.76,E2 -5322.76} C_VEL
LIN {X 0,Y 509.144,Z 432.653,A -85,B 0,C 180,E1 -5323.572,E2 -5323.572} C_VEL
LIN {X 0,Y 509.253,Z 429.743,A -85,B 0,C 180,E1 -5324.973,E2 -5324.973} C_VEL
LIN {X 0,Y 509.349,Z 425.264,A -85,B 0,C 180,E1 -5326.431,E2 -5326.431} C_VEL
LIN {X 0,Y 509.484,Z 420.178,A -85,B 0,C 180,E1 -5327.666,E2 -5327.666} C_VEL
LIN {X 0,Y 509.631,Z 413.695,A -85,B 0,C 180,E1 -5328.909,E2 -5328.909} C_VEL
LIN {X 0,Y 509.935,Z 405.461,A -85,B 0,C 180,E1 -5330.154,E2 -5330.154} C_VEL
LIN {X 0,Y 510.188,Z 396.959,A -85,B 0,C 180,E1 -5331.198,E2 -5331.198} C_VEL
LIN {X 0,Y 510.517,Z 387.604,A -85,B 0,C 180,E1 -5332.138,E2 -5332.138} C_VEL
LIN {X 0,Y 510.809,Z 377.315,A -85,B 0,C 180,E1 -5332.978,E2 -5332.978} C_VEL
LIN {X 0,Y 511.143,Z 365.951,A -85,B 0,C 180,E1 -5333.713,E2 -5333.713} C_VEL
LIN {X 0,Y 511.415,Z 353.223,A -85,B 0,C 180,E1 -5334.346,E2 -5334.346} C_VEL
LIN {X 0,Y 511.649,Z 340.556,A -85,B 0,C 180,E1 -5334.794,E2 -5334.794} C_VEL
LIN {X 0,Y 511.776,Z 326.718,A -85,B 0,C 180,E1 -5335.1,E2 -5335.1} C_VEL
LIN {X 0,Y 512.231,Z 234.719,A -85,B 0,C 180,E1 -5336.403,E2 -5336.403} C_VEL
LIN {X 0,Y 510.253,Z 224.364,A -85,B 0,C 180,E1 -5336.622,E2 -5336.622} C_VEL
LIN {X 0,Y 510.355,Z 210.475,A -85,B 0,C 180,E1 -5339.264,E2 -5339.264} C_VEL
LIN {X 0,Y 509.895,Z 205.974,A -85,B 0,C 180,E1 -5340.171,E2 -5340.171} C_VEL
LIN {X 0,Y 509.857,Z 205.972,A -85,B 0,C 180,E1 -5343.459,E2 -5343.459} C_VEL
LIN {X 0,Y 509.829,Z 205.983,A -85,B 0,C 180,E1 -5346.35,E2 -5346.35} C_VEL
LIN {X 0,Y 509.841,Z 205.976,A -85,B 0,C 180,E1 -5349.471,E2 -5349.471} C_VEL
LIN {X 0,Y 509.824,Z 205.981,A -85,B 0,C 180,E1 -5352.488,E2 -5352.488} C_VEL
LIN {X 0,Y 509.843,Z 205.973,A -85,B 0,C 180,E1 -5355.33,E2 -5355.33} C_VEL
LIN {X 0,Y 509.849,Z 205.975,A -85,B 0,C 180,E1 -5358.574,E2 -5358.574} C_VEL
LIN {X 0,Y 509.833,Z 205.979,A -85,B 0,C 180,E1 -5361.784,E2 -5361.784} C_VEL
LIN {X 0,Y 509.825,Z 205.975,A -85,B 0,C 180,E1 -5364.621,E2 -5364.621} C_VEL
LIN {X 0,Y 509.843,Z 205.976,A -85,B 0,C 180,E1 -5367.479,E2 -5367.479} C_VEL
LIN {X 0,Y 509.858,Z 205.974,A -85,B 0,C 180,E1 -5370.267,E2 -5370.267} C_VEL
LIN {X 0,Y 509.861,Z 205.968,A -85,B 0,C 180,E1 -5372.943,E2 -5372.943} C_VEL
LIN {X 0,Y 509.848,Z 205.978,A -85,B 0,C 180,E1 -5375.573,E2 -5375.573} C_VEL
LIN {X 0,Y 509.819,Z 205.978,A -85,B 0,C 180,E1 -5378.148,E2 -5378.148} C_VEL
LIN {X 0,Y 509.836,Z 205.97,A -85,B 0,C 180,E1 -5380.68,E2 -5380.68} C_VEL
LIN {X 0,Y 509.87,Z 205.972,A -85,B 0,C 180,E1 -5383.174,E2 -5383.174} C_VEL
LIN {X 0,Y 509.831,Z 205.981,A -85,B 0,C 180,E1 -5385.633,E2 -5385.633} C_VEL
LIN {X 0,Y 509.884,Z 205.967,A -85,B 0,C 180,E1 -5388.874,E2 -5388.874} C_VEL
LIN {X 0,Y 509.924,Z 205.962,A -85,B 0,C 180,E1 -5392.078,E2 -5392.078} C_VEL
LIN {X 0,Y 509.961,Z 205.956,A -85,B 0,C 180,E1 -5394.464,E2 -5394.464} C_VEL
LIN {X 0,Y 510.017,Z 205.951,A -85,B 0,C 180,E1 -5397.631,E2 -5397.631} C_VEL
LIN {X 0,Y 510.013,Z 205.951,A -85,B 0,C 180,E1 -5400,E2 -5400} C_VEL
LIN {X 0,Y 510.015,Z 205.95,A -85,B 0,C 180,E1 -5402.369,E2 -5402.369} C_VEL
LIN {X 0,Y 509.942,Z 205.962,A -85,B 0,C 180,E1 -5405.536,E2 -5405.536} C_VEL
LIN {X 0,Y 509.885,Z 205.964,A -85,B 0,C 180,E1 -5407.923,E2 -5407.923} C_VEL
LIN {X 0,Y 509.898,Z 205.969,A -85,B 0,C 180,E1 -5411.126,E2 -5411.126} C_VEL
LIN {X 0,Y 509.825,Z 205.976,A -85,B 0,C 180,E1 -5414.367,E2 -5414.367} C_VEL
LIN {X 0,Y 509.839,Z 205.978,A -85,B 0,C 180,E1 -5416.827,E2 -5416.827} C_VEL
LIN {X 0,Y 509.884,Z 205.968,A -85,B 0,C 180,E1 -5420.157,E2 -5420.157} C_VEL
LIN {X 0,Y 509.79,Z 205.979,A -85,B 0,C 180,E1 -5423.565,E2 -5423.565} C_VEL
LIN {X 0,Y 509.849,Z 205.973,A -85,B 0,C 180,E1 -5426.372,E2 -5426.372} C_VEL
LIN {X 0,Y 509.826,Z 205.977,A -85,B 0,C 180,E1 -5428.847,E2 -5428.847} C_VEL
LIN {X 0,Y 509.792,Z 205.979,A -85,B 0,C 180,E1 -5431.592,E2 -5431.592} C_VEL
LIN {X 0,Y 509.814,Z 205.981,A -85,B 0,C 180,E1 -5434.416,E2 -5434.416} C_VEL
LIN {X 0,Y 509.794,Z 205.974,A -85,B 0,C 180,E1 -5437.343,E2 -5437.343} C_VEL
LIN {X 0,Y 509.818,Z 205.981,A -85,B 0,C 180,E1 -5440.384,E2 -5440.384} C_VEL
LIN {X 0,Y 509.806,Z 205.977,A -85,B 0,C 180,E1 -5443.064,E2 -5443.064} C_VEL
LIN {X 0,Y 509.807,Z 205.979,A -85,B 0,C 180,E1 -5445.795,E2 -5445.795} C_VEL
LIN {X 0,Y 509.831,Z 205.977,A -85,B 0,C 180,E1 -5448.575,E2 -5448.575} C_VEL
LIN {X 0,Y 509.839,Z 205.977,A -85,B 0,C 180,E1 -5451.788,E2 -5451.788} C_VEL
LIN {X 0,Y 509.825,Z 205.976,A -85,B 0,C 180,E1 -5454.624,E2 -5454.624} C_VEL
LIN {X 0,Y 509.855,Z 205.973,A -85,B 0,C 180,E1 -5457.482,E2 -5457.482} C_VEL
LIN {X 0,Y 509.854,Z 205.977,A -85,B 0,C 180,E1 -5460.275,E2 -5460.275} C_VEL
LIN {X 0,Y 509.882,Z 205.973,A -85,B 0,C 180,E1 -5463.629,E2 -5463.629} C_VEL
LIN {X 0,Y 509.892,Z 206.032,A -85,B 0,C 180,E1 -5464.706,E2 -5464.706} C_VEL
LIN {X 0,Y 511.569,Z 215.564,A -85,B 0,C 180,E1 -5466.308,E2 -5466.308} C_VEL
LIN {X 0,Y 511.054,Z 234.431,A -85,B 0,C 180,E1 -5469.25,E2 -5469.25} C_VEL
LIN {X 0,Y 510.545,Z 254.792,A -85,B 0,C 180,E1 -5472.372,E2 -5472.372} C_VEL
LIN {X 0,Y 510.234,Z 268.208,A -85,B 0,C 180,E1 -5474.405,E2 -5474.405} C_VEL
LIN {X 0,Y 512.184,Z 281.393,A -85,B 0,C 180,E1 -5474.658,E2 -5474.658} C_VEL
LIN {X 0,Y 511.711,Z 376.675,A -85,B 0,C 180,E1 -5476.017,E2 -5476.017} C_VEL
LIN {X 0,Y 511.439,Z 390.034,A -85,B 0,C 180,E1 -5476.364,E2 -5476.364} C_VEL
LIN {X 0,Y 511.108,Z 402.251,A -85,B 0,C 180,E1 -5476.836,E2 -5476.836} C_VEL
LIN {X 0,Y 510.848,Z 413.753,A -85,B 0,C 180,E1 -5477.434,E2 -5477.434} C_VEL
LIN {X 0,Y 510.5,Z 424.93,A -85,B 0,C 180,E1 -5478.183,E2 -5478.183} C_VEL
LIN {X 0,Y 510.21,Z 435.64,A -85,B 0,C 180,E1 -5479.082,E2 -5479.082} C_VEL
LIN {X 0,Y 509.861,Z 445.29,A -85,B 0,C 180,E1 -5480.078,E2 -5480.078} C_VEL
LIN {X 0,Y 509.656,Z 453.208,A -85,B 0,C 180,E1 -5481.075,E2 -5481.075} C_VEL
LIN {X 0,Y 509.435,Z 460.942,A -85,B 0,C 180,E1 -5482.269,E2 -5482.269} C_VEL
LIN {X 0,Y 509.309,Z 468.075,A -85,B 0,C 180,E1 -5483.661,E2 -5483.661} C_VEL
LIN {X 0,Y 509.241,Z 472.822,A -85,B 0,C 180,E1 -5484.852,E2 -5484.852} C_VEL
LIN {X 0,Y 509.246,Z 476.453,A -85,B 0,C 180,E1 -5486.042,E2 -5486.042} C_VEL
LIN {X 0,Y 509.201,Z 478.324,A -85,B 0,C 180,E1 -5486.834,E2 -5486.834} C_VEL
LIN {X 0,Y 509.19,Z 479.728,A -85,B 0,C 180,E1 -5487.626,E2 -5487.626} C_VEL
LIN {X 0,Y 509.08,Z 481.34,A -85,B 0,C 180,E1 -5489.208,E2 -5489.208} C_VEL
LIN {X 0,Y 509.078,Z 481.56,A -85,B 0,C 180,E1 -5489.999,E2 -5489.999} C_VEL
LIN {X 0,Y 509.112,Z 480.74,A -85,B 0,C 180,E1 -5491.58,E2 -5491.58} C_VEL
LIN {X 0,Y 509.189,Z 479.747,A -85,B 0,C 180,E1 -5492.371,E2 -5492.371} C_VEL
LIN {X 0,Y 509.2,Z 478.348,A -85,B 0,C 180,E1 -5493.163,E2 -5493.163} C_VEL
LIN {X 0,Y 509.203,Z 475.403,A -85,B 0,C 180,E1 -5494.352,E2 -5494.352} C_VEL
LIN {X 0,Y 509.283,Z 471.419,A -85,B 0,C 180,E1 -5495.541,E2 -5495.541} C_VEL
LIN {X 0,Y 509.351,Z 465.744,A -85,B 0,C 180,E1 -5496.843,E2 -5496.843} C_VEL
LIN {X 0,Y 509.512,Z 458.591,A -85,B 0,C 180,E1 -5498.126,E2 -5498.126} C_VEL
LIN {X 0,Y 509.73,Z 450.283,A -85,B 0,C 180,E1 -5499.321,E2 -5499.321} C_VEL
LIN {X 0,Y 509.97,Z 441.77,A -85,B 0,C 180,E1 -5500.318,E2 -5500.318} C_VEL
LIN {X 0,Y 510.348,Z 431.257,A -85,B 0,C 180,E1 -5501.314,E2 -5501.314} C_VEL
LIN {X 0,Y 510.668,Z 420.911,A -85,B 0,C 180,E1 -5502.109,E2 -5502.109} C_VEL
LIN {X 0,Y 510.98,Z 409.463,A -85,B 0,C 180,E1 -5502.811,E2 -5502.811} C_VEL
LIN {X 0,Y 511.256,Z 397.773,A -85,B 0,C 180,E1 -5503.36,E2 -5503.36} C_VEL
LIN {X 0,Y 511.552,Z 384.315,A -85,B 0,C 180,E1 -5503.807,E2 -5503.807} C_VEL
LIN {X 0,Y 511.776,Z 371.02,A -85,B 0,C 180,E1 -5504.08,E2 -5504.08} C_VEL
LIN {X 0,Y 512.01,Z 280.455,A -85,B 0,C 180,E1 -5505.361,E2 -5505.361} C_VEL
LIN {X 0,Y 510.25,Z 268.247,A -85,B 0,C 180,E1 -5505.605,E2 -5505.605} C_VEL
LIN {X 0,Y 510.724,Z 248.208,A -85,B 0,C 180,E1 -5508.656,E2 -5508.656} C_VEL
LIN {X 0,Y 511.217,Z 227.891,A -85,B 0,C 180,E1 -5511.785,E2 -5511.785} C_VEL
LIN {X 0,Y 511.595,Z 215.65,A -85,B 0,C 180,E1 -5513.688,E2 -5513.688} C_VEL
LIN {X 0,Y 509.877,Z 205.974,A -85,B 0,C 180,E1 -5515.319,E2 -5515.319} C_VEL
LIN {X 0,Y 509.883,Z 205.976,A -85,B 0,C 180,E1 -5518.097,E2 -5518.097} C_VEL
LIN {X 0,Y 509.828,Z 205.974,A -85,B 0,C 180,E1 -5521.276,E2 -5521.276} C_VEL
LIN {X 0,Y 509.841,Z 205.978,A -85,B 0,C 180,E1 -5524.2,E2 -5524.2} C_VEL
LIN {X 0,Y 509.794,Z 205.979,A -85,B 0,C 180,E1 -5527.337,E2 -5527.337} C_VEL
LIN {X 0,Y 509.81,Z 205.978,A -85,B 0,C 180,E1 -5530.378,E2 -5530.378} C_VEL
LIN {X 0,Y 509.792,Z 205.978,A -85,B 0,C 180,E1 -5533.058,E2 -5533.058} C_VEL
LIN {X 0,Y 509.798,Z 205.986,A -85,B 0,C 180,E1 -5535.788,E2 -5535.788} C_VEL
LIN {X 0,Y 509.837,Z 205.973,A -85,B 0,C 180,E1 -5538.572,E2 -5538.572} C_VEL
LIN {X 0,Y 509.817,Z 205.983,A -85,B 0,C 180,E1 -5541.782,E2 -5541.782} C_VEL
LIN {X 0,Y 509.804,Z 205.977,A -85,B 0,C 180,E1 -5544.62,E2 -5544.62} C_VEL
LIN {X 0,Y 509.829,Z 205.98,A -85,B 0,C 180,E1 -5547.478,E2 -5547.478} C_VEL
LIN {X 0,Y 509.835,Z 205.973,A -85,B 0,C 180,E1 -5550.266,E2 -5550.266} C_VEL
LIN {X 0,Y 509.838,Z 205.974,A -85,B 0,C 180,E1 -5552.942,E2 -5552.942} C_VEL
LIN {X 0,Y 509.842,Z 205.979,A -85,B 0,C 180,E1 -5555.573,E2 -5555.573} C_VEL
LIN {X 0,Y 509.813,Z 205.976,A -85,B 0,C 180,E1 -5558.148,E2 -5558.148} C_VEL
LIN {X 0,Y 509.812,Z 205.976,A -85,B 0,C 180,E1 -5560.68,E2 -5560.68} C_VEL
LIN {X 0,Y 509.846,Z 205.978,A -85,B 0,C 180,E1 -5563.173,E2 -5563.173} C_VEL
LIN {X 0,Y 509.818,Z 205.979,A -85,B 0,C 180,E1 -5565.633,E2 -5565.633} C_VEL
LIN {X 0,Y 509.884,Z 205.967,A -85,B 0,C 180,E1 -5568.099,E2 -5568.099} C_VEL
LIN {X 0,Y 509.89,Z 205.974,A -85,B 0,C 180,E1 -5571.279,E2 -5571.279} C_VEL
LIN {X 0,Y 509.932,Z 205.963,A -85,B 0,C 180,E1 -5573.67,E2 -5573.67} C_VEL
LIN {X 0,Y 509.927,Z 205.966,A -85,B 0,C 180,E1 -5576.84,E2 -5576.84} C_VEL
LIN {X 0,Y 509.99,Z 205.953,A -85,B 0,C 180,E1 -5580,E2 -5580} C_VEL
LIN {X 0,Y 509.993,Z 205.954,A -85,B 0,C 180,E1 -5582.369,E2 -5582.369} C_VEL
LIN {X 0,Y 509.917,Z 205.964,A -85,B 0,C 180,E1 -5586.33,E2 -5586.33} C_VEL
LIN {X 0,Y 509.86,Z 205.976,A -85,B 0,C 180,E1 -5588.721,E2 -5588.721} C_VEL
LIN {X 0,Y 509.893,Z 205.966,A -85,B 0,C 180,E1 -5591.932,E2 -5591.932} C_VEL
LIN {X 0,Y 509.836,Z 205.975,A -85,B 0,C 180,E1 -5595.244,E2 -5595.244} C_VEL
LIN {X 0,Y 509.833,Z 205.974,A -85,B 0,C 180,E1 -5598.003,E2 -5598.003} C_VEL
LIN {X 0,Y 509.803,Z 205.981,A -85,B 0,C 180,E1 -5601.004,E2 -5601.004} C_VEL
LIN {X 0,Y 509.797,Z 205.977,A -85,B 0,C 180,E1 -5603.565,E2 -5603.565} C_VEL
LIN {X 0,Y 509.863,Z 205.975,A -85,B 0,C 180,E1 -5606.382,E2 -5606.382} C_VEL
LIN {X 0,Y 509.843,Z 205.976,A -85,B 0,C 180,E1 -5608.847,E2 -5608.847} C_VEL
LIN {X 0,Y 509.78,Z 205.98,A -85,B 0,C 180,E1 -5611.593,E2 -5611.593} C_VEL
LIN {X 0,Y 509.811,Z 205.984,A -85,B 0,C 180,E1 -5614.417,E2 -5614.417} C_VEL
LIN {X 0,Y 509.778,Z 205.98,A -85,B 0,C 180,E1 -5617.344,E2 -5617.344} C_VEL
LIN {X 0,Y 509.823,Z 205.983,A -85,B 0,C 180,E1 -5620.384,E2 -5620.384} C_VEL
LIN {X 0,Y 509.805,Z 205.977,A -85,B 0,C 180,E1 -5623.068,E2 -5623.068} C_VEL
LIN {X 0,Y 509.799,Z 205.98,A -85,B 0,C 180,E1 -5625.796,E2 -5625.796} C_VEL
LIN {X 0,Y 509.83,Z 205.977,A -85,B 0,C 180,E1 -5628.579,E2 -5628.579} C_VEL
LIN {X 0,Y 509.826,Z 205.978,A -85,B 0,C 180,E1 -5631.791,E2 -5631.791} C_VEL
LIN {X 0,Y 509.806,Z 205.978,A -85,B 0,C 180,E1 -5633.773,E2 -5633.773} C_VEL
LIN {X 0,Y 509.143,Z 206.063,A -85,B 0,C 180,E1 -5634.433,E2 -5634.433} C_VEL
LIN {X 0,Y 506.325,Z 206.412,A -85,B 0,C 180,E1 -5635.505,E2 -5635.505} C_VEL
LIN {X 0,Y 503.932,Z 206.712,A -85,B 0,C 180,E1 -5636.368,E2 -5636.368} C_VEL
LIN {X 0,Y 502.883,Z 206.839,A -85,B 0,C 180,E1 -5637.034,E2 -5637.034} C_VEL
LIN {X 0,Y 502.786,Z 206.851,A -85,B 0,C 180,E1 -5637.26,E2 -5637.26} C_VEL
LIN {X 0,Y 502.799,Z 206.857,A -85,B 0,C 180,E1 -5640.069,E2 -5640.069} C_VEL
LIN {X 0,Y 502.818,Z 206.848,A -85,B 0,C 180,E1 -5642.537,E2 -5642.537} C_VEL
LIN {X 0,Y 502.792,Z 206.852,A -85,B 0,C 180,E1 -5645.309,E2 -5645.309} C_VEL
LIN {X 0,Y 502.771,Z 206.861,A -85,B 0,C 180,E1 -5647.83,E2 -5647.83} C_VEL
LIN {X 0,Y 502.813,Z 206.849,A -85,B 0,C 180,E1 -5650.403,E2 -5650.403} C_VEL
LIN {X 0,Y 502.804,Z 206.849,A -85,B 0,C 180,E1 -5652.934,E2 -5652.934} C_VEL
LIN {X 0,Y 502.83,Z 206.85,A -85,B 0,C 180,E1 -5655.432,E2 -5655.432} C_VEL
LIN {X 0,Y 502.876,Z 206.842,A -85,B 0,C 180,E1 -5658.719,E2 -5658.719} C_VEL
LIN {X 0,Y 502.931,Z 206.936,A -85,B 0,C 180,E1 -5661.793,E2 -5661.793} C_VEL
LIN {X 0,Y 503.486,Z 212.917,A -85,B 0,C 180,E1 -5662.987,E2 -5662.987} C_VEL
LIN {X 0,Y 503.256,Z 223.273,A -85,B 0,C 180,E1 -5664.995,E2 -5664.995} C_VEL
LIN {X 0,Y 503.14,Z 224.592,A -85,B 0,C 180,E1 -5665.245,E2 -5665.245} C_VEL
LIN {X 0,Y 505.446,Z 235.718,A -85,B 0,C 180,E1 -5665.49,E2 -5665.49} C_VEL
LIN {X 0,Y 504.846,Z 331.898,A -85,B 0,C 180,E1 -5666.885,E2 -5666.885} C_VEL
LIN {X 0,Y 504.668,Z 345.536,A -85,B 0,C 180,E1 -5667.258,E2 -5667.258} C_VEL
LIN {X 0,Y 504.417,Z 357.817,A -85,B 0,C 180,E1 -5667.756,E2 -5667.756} C_VEL
LIN {X 0,Y 504.13,Z 369.582,A -85,B 0,C 180,E1 -5668.404,E2 -5668.404} C_VEL
LIN {X 0,Y 503.683,Z 380.902,A -85,B 0,C 180,E1 -5669.202,E2 -5669.202} C_VEL
LIN {X 0,Y 503.351,Z 391.092,A -85,B 0,C 180,E1 -5670.101,E2 -5670.101} C_VEL
LIN {X 0,Y 503.102,Z 399.438,A -85,B 0,C 180,E1 -5671.002,E2 -5671.002} C_VEL
LIN {X 0,Y 502.752,Z 408.528,A -85,B 0,C 180,E1 -5672.204,E2 -5672.204} C_VEL
LIN {X 0,Y 502.535,Z 415.844,A -85,B 0,C 180,E1 -5673.409,E2 -5673.409} C_VEL
LIN {X 0,Y 502.387,Z 422.605,A -85,B 0,C 180,E1 -5674.816,E2 -5674.816} C_VEL
LIN {X 0,Y 502.276,Z 427.079,A -85,B 0,C 180,E1 -5676.025,E2 -5676.025} C_VEL
LIN {X 0,Y 502.195,Z 430.491,A -85,B 0,C 180,E1 -5677.236,E2 -5677.236} C_VEL
LIN {X 0,Y 502.119,Z 432.192,A -85,B 0,C 180,E1 -5678.047,E2 -5678.047} C_VEL
LIN {X 0,Y 502.071,Z 433.49,A -85,B 0,C 180,E1 -5678.858,E2 -5678.858} C_VEL
LIN {X 0,Y 502.035,Z 434.396,A -85,B 0,C 180,E1 -5679.671,E2 -5679.671} C_VEL
LIN {X 0,Y 502.092,Z 434.872,A -85,B 0,C 180,E1 -5680.485,E2 -5680.485} C_VEL
LIN {X 0,Y 502.107,Z 434.889,A -85,B 0,C 180,E1 -5681.537,E2 -5681.537} C_VEL
LIN {X 0,Y 502.047,Z 433.886,A -85,B 0,C 180,E1 -5682.943,E2 -5682.943} C_VEL
LIN {X 0,Y 502.072,Z 432.705,A -85,B 0,C 180,E1 -5683.767,E2 -5683.767} C_VEL
LIN {X 0,Y 502.184,Z 429.987,A -85,B 0,C 180,E1 -5685.061,E2 -5685.061} C_VEL
LIN {X 0,Y 502.264,Z 426.487,A -85,B 0,C 180,E1 -5686.251,E2 -5686.251} C_VEL
LIN {X 0,Y 502.395,Z 421.648,A -85,B 0,C 180,E1 -5687.503,E2 -5687.503} C_VEL
LIN {X 0,Y 502.573,Z 415.449,A -85,B 0,C 180,E1 -5688.761,E2 -5688.761} C_VEL
LIN {X 0,Y 502.87,Z 407.655,A -85,B 0,C 180,E1 -5690.023,E2 -5690.023} C_VEL
LIN {X 0,Y 503.127,Z 399.676,A -85,B 0,C 180,E1 -5691.067,E2 -5691.067} C_VEL
LIN {X 0,Y 503.472,Z 389.551,A -85,B 0,C 180,E1 -5692.141,E2 -5692.141} C_VEL
LIN {X 0,Y 503.791,Z 379.658,A -85,B 0,C 180,E1 -5692.991,E2 -5692.991} C_VEL
LIN {X 0,Y 504.163,Z 368.933,A -85,B 0,C 180,E1 -5693.735,E2 -5693.735} C_VEL
LIN {X 0,Y 504.449,Z 357.035,A -85,B 0,C 180,E1 -5694.376,E2 -5694.376} C_VEL
LIN {X 0,Y 504.698,Z 344.43,A -85,B 0,C 180,E1 -5694.875,E2 -5694.875} C_VEL
LIN {X 0,Y 504.862,Z 331.431,A -85,B 0,C 180,E1 -5695.221,E2 -5695.221} C_VEL
LIN {X 0,Y 505.467,Z 236.052,A -85,B 0,C 180,E1 -5696.603,E2 -5696.603} C_VEL
LIN {X 0,Y 503.311,Z 224.606,A -85,B 0,C 180,E1 -5696.854,E2 -5696.854} C_VEL
LIN {X 0,Y 503.351,Z 210.213,A -85,B 0,C 180,E1 -5699.619,E2 -5699.619} C_VEL
LIN {X 0,Y 502.834,Z 206.853,A -85,B 0,C 180,E1 -5700.324,E2 -5700.324} C_VEL
LIN {X 0,Y 502.828,Z 206.849,A -85,B 0,C 180,E1 -5703.03,E2 -5703.03} C_VEL
LIN {X 0,Y 502.777,Z 206.858,A -85,B 0,C 180,E1 -5705.949,E2 -5705.949} C_VEL
LIN {X 0,Y 502.801,Z 206.854,A -85,B 0,C 180,E1 -5708.973,E2 -5708.973} C_VEL
LIN {X 0,Y 502.817,Z 206.85,A -85,B 0,C 180,E1 -5711.063,E2 -5711.063} C_VEL
LIN {X 0,Y 502.788,Z 206.856,A -85,B 0,C 180,E1 -5714.53,E2 -5714.53} C_VEL
LIN {X 0,Y 502.815,Z 206.853,A -85,B 0,C 180,E1 -5717.862,E2 -5717.862} C_VEL
LIN {X 0,Y 502.792,Z 206.851,A -85,B 0,C 180,E1 -5721.023,E2 -5721.023} C_VEL
LIN {X 0,Y 502.765,Z 206.86,A -85,B 0,C 180,E1 -5724.165,E2 -5724.165} C_VEL
LIN {X 0,Y 502.811,Z 206.848,A -85,B 0,C 180,E1 -5726.991,E2 -5726.991} C_VEL
LIN {X 0,Y 502.807,Z 206.855,A -85,B 0,C 180,E1 -5730.06,E2 -5730.06} C_VEL
LIN {X 0,Y 502.81,Z 206.847,A -85,B 0,C 180,E1 -5732.532,E2 -5732.532} C_VEL
LIN {X 0,Y 502.804,Z 206.852,A -85,B 0,C 180,E1 -5735.296,E2 -5735.296} C_VEL
LIN {X 0,Y 502.782,Z 206.858,A -85,B 0,C 180,E1 -5737.826,E2 -5737.826} C_VEL
LIN {X 0,Y 502.796,Z 206.848,A -85,B 0,C 180,E1 -5740.399,E2 -5740.399} C_VEL
LIN {X 0,Y 502.816,Z 206.849,A -85,B 0,C 180,E1 -5742.931,E2 -5742.931} C_VEL
LIN {X 0,Y 502.813,Z 206.852,A -85,B 0,C 180,E1 -5745.428,E2 -5745.428} C_VEL
LIN {X 0,Y 502.848,Z 206.843,A -85,B 0,C 180,E1 -5748.716,E2 -5748.716} C_VEL
LIN {X 0,Y 502.872,Z 206.842,A -85,B 0,C 180,E1 -5751.966,E2 -5751.966} C_VEL
LIN {X 0,Y 502.916,Z 206.833,A -85,B 0,C 180,E1 -5754.386,E2 -5754.386} C_VEL
LIN {X 0,Y 502.987,Z 206.827,A -85,B 0,C 180,E1 -5757.598,E2 -5757.598} C_VEL
LIN {X 0,Y 502.985,Z 206.827,A -85,B 0,C 180,E1 -5760,E2 -5760} C_VEL
LIN {X 0,Y 502.985,Z 206.825,A -85,B 0,C 180,E1 -5762.402,E2 -5762.402} C_VEL
LIN {X 0,Y 502.896,Z 206.839,A -85,B 0,C 180,E1 -5765.614,E2 -5765.614} C_VEL
LIN {X 0,Y 502.845,Z 206.841,A -85,B 0,C 180,E1 -5768.034,E2 -5768.034} C_VEL
LIN {X 0,Y 502.866,Z 206.843,A -85,B 0,C 180,E1 -5771.283,E2 -5771.283} C_VEL
LIN {X 0,Y 502.808,Z 206.852,A -85,B 0,C 180,E1 -5774.572,E2 -5774.572} C_VEL
LIN {X 0,Y 502.789,Z 206.849,A -85,B 0,C 180,E1 -5777.91,E2 -5777.91} C_VEL
LIN {X 0,Y 502.799,Z 206.855,A -85,B 0,C 180,E1 -5780.537,E2 -5780.537} C_VEL
LIN {X 0,Y 502.757,Z 206.859,A -85,B 0,C 180,E1 -5783.042,E2 -5783.042} C_VEL
LIN {X 0,Y 502.766,Z 206.851,A -85,B 0,C 180,E1 -5785.68,E2 -5785.68} C_VEL
LIN {X 0,Y 502.771,Z 206.859,A -85,B 0,C 180,E1 -5788.377,E2 -5788.377} C_VEL
LIN {X 0,Y 502.768,Z 206.855,A -85,B 0,C 180,E1 -5791.145,E2 -5791.145} C_VEL
LIN {X 0,Y 502.764,Z 206.854,A -85,B 0,C 180,E1 -5793.997,E2 -5793.997} C_VEL
LIN {X 0,Y 502.755,Z 206.852,A -85,B 0,C 180,E1 -5797.179,E2 -5797.179} C_VEL
LIN {X 0,Y 502.764,Z 206.853,A -85,B 0,C 180,E1 -5800.018,E2 -5800.018} C_VEL
LIN {X 0,Y 502.787,Z 206.859,A -85,B 0,C 180,E1 -5802.201,E2 -5802.201} C_VEL
LIN {X 0,Y 502.771,Z 206.853,A -85,B 0,C 180,E1 -5805.472,E2 -5805.472} C_VEL
LIN {X 0,Y 502.782,Z 206.856,A -85,B 0,C 180,E1 -5807.862,E2 -5807.862} C_VEL
LIN {X 0,Y 502.782,Z 206.852,A -85,B 0,C 180,E1 -5811.025,E2 -5811.025} C_VEL
LIN {X 0,Y 502.769,Z 206.859,A -85,B 0,C 180,E1 -5814.17,E2 -5814.17} C_VEL
LIN {X 0,Y 502.827,Z 206.846,A -85,B 0,C 180,E1 -5816.995,E2 -5816.995} C_VEL
LIN {X 0,Y 502.811,Z 206.856,A -85,B 0,C 180,E1 -5820.066,E2 -5820.066} C_VEL
LIN {X 0,Y 502.842,Z 206.85,A -85,B 0,C 180,E1 -5823.444,E2 -5823.444} C_VEL
LIN {X 0,Y 502.868,Z 207.003,A -85,B 0,C 180,E1 -5824.521,E2 -5824.521} C_VEL
LIN {X 0,Y 504.622,Z 216.683,A -85,B 0,C 180,E1 -5826.179,E2 -5826.179} C_VEL
LIN {X 0,Y 504.141,Z 234.336,A -85,B 0,C 180,E1 -5828.979,E2 -5828.979} C_VEL
LIN {X 0,Y 503.565,Z 254.489,A -85,B 0,C 180,E1 -5832.119,E2 -5832.119} C_VEL
LIN {X 0,Y 503.208,Z 267.867,A -85,B 0,C 180,E1 -5834.179,E2 -5834.179} C_VEL
LIN {X 0,Y 505.339,Z 282.563,A -85,B 0,C 180,E1 -5834.465,E2 -5834.465} C_VEL
LIN {X 0,Y 504.831,Z 376.346,A -85,B 0,C 180,E1 -5835.822,E2 -5835.822} C_VEL
LIN {X 0,Y 504.547,Z 389.696,A -85,B 0,C 180,E1 -5836.174,E2 -5836.174} C_VEL
LIN {X 0,Y 504.151,Z 403.035,A -85,B 0,C 180,E1 -5836.702,E2 -5836.702} C_VEL
LIN {X 0,Y 503.864,Z 415.433,A -85,B 0,C 180,E1 -5837.386,E2 -5837.386} C_VEL
LIN {X 0,Y 503.438,Z 427.183,A -85,B 0,C 180,E1 -5838.219,E2 -5838.219} C_VEL
LIN {X 0,Y 503.155,Z 437.428,A -85,B 0,C 180,E1 -5839.13,E2 -5839.13} C_VEL
LIN {X 0,Y 502.789,Z 446.64,A -85,B 0,C 180,E1 -5840.14,E2 -5840.14} C_VEL
LIN {X 0,Y 502.535,Z 455.624,A -85,B 0,C 180,E1 -5841.353,E2 -5841.353} C_VEL
LIN {X 0,Y 502.332,Z 462.857,A -85,B 0,C 180,E1 -5842.563,E2 -5842.563} C_VEL
LIN {X 0,Y 502.236,Z 467.741,A -85,B 0,C 180,E1 -5843.572,E2 -5843.572} C_VEL
LIN {X 0,Y 502.172,Z 472.491,A -85,B 0,C 180,E1 -5844.78,E2 -5844.78} C_VEL
LIN {X 0,Y 502.14,Z 476.121,A -85,B 0,C 180,E1 -5845.986,E2 -5845.986} C_VEL
LIN {X 0,Y 502.12,Z 477.995,A -85,B 0,C 180,E1 -5846.789,E2 -5846.789} C_VEL
LIN {X 0,Y 502.121,Z 479.401,A -85,B 0,C 180,E1 -5847.592,E2 -5847.592} C_VEL
LIN {X 0,Y 501.996,Z 481.013,A -85,B 0,C 180,E1 -5849.196,E2 -5849.196} C_VEL
LIN {X 0,Y 501.992,Z 481.234,A -85,B 0,C 180,E1 -5849.998,E2 -5849.998} C_VEL
LIN {X 0,Y 502.036,Z 480.415,A -85,B 0,C 180,E1 -5851.603,E2 -5851.603} C_VEL
LIN {X 0,Y 502.12,Z 479.422,A -85,B 0,C 180,E1 -5852.405,E2 -5852.405} C_VEL
LIN {X 0,Y 502.12,Z 478.022,A -85,B 0,C 180,E1 -5853.208,E2 -5853.208} C_VEL
LIN {X 0,Y 502.101,Z 475.076,A -85,B 0,C 180,E1 -5854.413,E2 -5854.413} C_VEL
LIN {X 0,Y 502.199,Z 471.092,A -85,B 0,C 180,E1 -5855.62,E2 -5855.62} C_VEL
LIN {X 0,Y 502.289,Z 465.063,A -85,B 0,C 180,E1 -5857.01,E2 -5857.01} C_VEL
LIN {X 0,Y 502.459,Z 458.263,A -85,B 0,C 180,E1 -5858.241,E2 -5858.241} C_VEL
LIN {X 0,Y 502.695,Z 449.954,A -85,B 0,C 180,E1 -5859.453,E2 -5859.453} C_VEL
LIN {X 0,Y 502.962,Z 441.44,A -85,B 0,C 180,E1 -5860.463,E2 -5860.463} C_VEL
LIN {X 0,Y 503.367,Z 430.926,A -85,B 0,C 180,E1 -5861.473,E2 -5861.473} C_VEL
LIN {X 0,Y 503.681,Z 420.577,A -85,B 0,C 180,E1 -5862.279,E2 -5862.279} C_VEL
LIN {X 0,Y 504.024,Z 409.127,A -85,B 0,C 180,E1 -5862.991,E2 -5862.991} C_VEL
LIN {X 0,Y 504.345,Z 397.434,A -85,B 0,C 180,E1 -5863.546,E2 -5863.546} C_VEL
LIN {X 0,Y 504.663,Z 383.97,A -85,B 0,C 180,E1 -5864,E2 -5864} C_VEL
LIN {X 0,Y 504.902,Z 370.647,A -85,B 0,C 180,E1 -5864.276,E2 -5864.276} C_VEL
LIN {X 0,Y 505.192,Z 281.419,A -85,B 0,C 180,E1 -5865.554,E2 -5865.554} C_VEL
LIN {X 0,Y 503.227,Z 267.978,A -85,B 0,C 180,E1 -5865.818,E2 -5865.818} C_VEL
LIN {X 0,Y 503.733,Z 249.202,A -85,B 0,C 180,E1 -5868.713,E2 -5868.713} C_VEL
LIN {X 0,Y 504.258,Z 228.856,A -85,B 0,C 180,E1 -5871.886,E2 -5871.886} C_VEL
LIN {X 0,Y 504.607,Z 216.595,A -85,B 0,C 180,E1 -5873.818,E2 -5873.818} C_VEL
LIN {X 0,Y 502.862,Z 206.848,A -85,B 0,C 180,E1 -5875.476,E2 -5875.476} C_VEL
LIN {X 0,Y 502.825,Z 206.854,A -85,B 0,C 180,E1 -5878.369,E2 -5878.369} C_VEL
LIN {X 0,Y 502.775,Z 206.854,A -85,B 0,C 180,E1 -5881.495,E2 -5881.495} C_VEL
LIN {X 0,Y 502.786,Z 206.854,A -85,B 0,C 180,E1 -5884.441,E2 -5884.441} C_VEL
LIN {X 0,Y 502.756,Z 206.855,A -85,B 0,C 180,E1 -5887.174,E2 -5887.174} C_VEL
LIN {X 0,Y 502.761,Z 206.861,A -85,B 0,C 180,E1 -5890.011,E2 -5890.011} C_VEL
LIN {X 0,Y 502.773,Z 206.857,A -85,B 0,C 180,E1 -5892.195,E2 -5892.195} C_VEL
LIN {X 0,Y 502.767,Z 206.857,A -85,B 0,C 180,E1 -5895.464,E2 -5895.464} C_VEL
LIN {X 0,Y 502.803,Z 206.856,A -85,B 0,C 180,E1 -5897.861,E2 -5897.861} C_VEL
LIN {X 0,Y 502.783,Z 206.852,A -85,B 0,C 180,E1 -5901.022,E2 -5901.022} C_VEL
LIN {X 0,Y 502.744,Z 206.858,A -85,B 0,C 180,E1 -5904.164,E2 -5904.164} C_VEL
LIN {X 0,Y 502.79,Z 206.851,A -85,B 0,C 180,E1 -5906.99,E2 -5906.99} C_VEL
LIN {X 0,Y 502.784,Z 206.853,A -85,B 0,C 180,E1 -5910.058,E2 -5910.058} C_VEL
LIN {X 0,Y 502.787,Z 206.851,A -85,B 0,C 180,E1 -5912.53,E2 -5912.53} C_VEL
LIN {X 0,Y 502.787,Z 206.857,A -85,B 0,C 180,E1 -5915.293,E2 -5915.293} C_VEL
LIN {X 0,Y 502.774,Z 206.856,A -85,B 0,C 180,E1 -5917.826,E2 -5917.826} C_VEL
LIN {X 0,Y 502.777,Z 206.852,A -85,B 0,C 180,E1 -5920.398,E2 -5920.398} C_VEL
LIN {X 0,Y 502.792,Z 206.853,A -85,B 0,C 180,E1 -5922.93,E2 -5922.93} C_VEL
LIN {X 0,Y 502.795,Z 206.857,A -85,B 0,C 180,E1 -5925.428,E2 -5925.428} C_VEL
LIN {X 0,Y 502.844,Z 206.846,A -85,B 0,C 180,E1 -5928.716,E2 -5928.716} C_VEL
LIN {X 0,Y 502.859,Z 206.842,A -85,B 0,C 180,E1 -5931.966,E2 -5931.966} C_VEL
LIN {X 0,Y 502.905,Z 206.836,A -85,B 0,C 180,E1 -5934.386,E2 -5934.386} C_VEL
LIN {X 0,Y 502.967,Z 206.83,A -85,B 0,C 180,E1 -5937.598,E2 -5937.598} C_VEL
LIN {X 0,Y 502.961,Z 206.829,A -85,B 0,C 180,E1 -5940,E2 -5940} C_VEL
LIN {X 0,Y 502.963,Z 206.83,A -85,B 0,C 180,E1 -5942.403,E2 -5942.403} C_VEL
LIN {X 0,Y 502.887,Z 206.839,A -85,B 0,C 180,E1 -5945.614,E2 -5945.614} C_VEL
LIN {X 0,Y 502.842,Z 206.844,A -85,B 0,C 180,E1 -5948.034,E2 -5948.034} C_VEL
LIN {X 0,Y 502.843,Z 206.847,A -85,B 0,C 180,E1 -5951.284,E2 -5951.284} C_VEL
LIN {X 0,Y 502.795,Z 206.855,A -85,B 0,C 180,E1 -5954.572,E2 -5954.572} C_VEL
LIN {X 0,Y 502.807,Z 206.848,A -85,B 0,C 180,E1 -5957.909,E2 -5957.909} C_VEL
LIN {X 0,Y 502.776,Z 206.859,A -85,B 0,C 180,E1 -5960.539,E2 -5960.539} C_VEL
LIN {X 0,Y 502.753,Z 206.858,A -85,B 0,C 180,E1 -5963.043,E2 -5963.043} C_VEL
LIN {X 0,Y 502.791,Z 206.85,A -85,B 0,C 180,E1 -5965.678,E2 -5965.678} C_VEL
LIN {X 0,Y 502.796,Z 206.856,A -85,B 0,C 180,E1 -5968.376,E2 -5968.376} C_VEL
LIN {X 0,Y 502.751,Z 206.855,A -85,B 0,C 180,E1 -5971.503,E2 -5971.503} C_VEL
LIN {X 0,Y 502.764,Z 206.863,A -85,B 0,C 180,E1 -5974.448,E2 -5974.448} C_VEL
LIN {X 0,Y 502.741,Z 206.857,A -85,B 0,C 180,E1 -5977.182,E2 -5977.182} C_VEL
LIN {X 0,Y 502.779,Z 206.856,A -85,B 0,C 180,E1 -5980.016,E2 -5980.016} C_VEL
LIN {X 0,Y 502.788,Z 206.858,A -85,B 0,C 180,E1 -5982.206,E2 -5982.206} C_VEL
LIN {X 0,Y 502.769,Z 206.853,A -85,B 0,C 180,E1 -5985.472,E2 -5985.472} C_VEL
LIN {X 0,Y 502.793,Z 206.85,A -85,B 0,C 180,E1 -5988.938,E2 -5988.938} C_VEL
LIN {X 0,Y 502.769,Z 206.861,A -85,B 0,C 180,E1 -5992.05,E2 -5992.05} C_VEL
LIN {X 0,Y 502.786,Z 206.851,A -85,B 0,C 180,E1 -5995.039,E2 -5995.039} C_VEL
LIN {X 0,Y 502.786,Z 206.851,A -85,B 0,C 180,E1 -5997.26,E2 -5997.26} C_VEL
LIN {X 0,Y 502.087,Z 206.945,A -85,B 0,C 180,E1 -5997.929,E2 -5997.929} C_VEL
LIN {X 0,Y 499.223,Z 207.299,A -85,B 0,C 180,E1 -5999.014,E2 -5999.014} C_VEL
LIN {X 0,Y 496.829,Z 207.6,A -85,B 0,C 180,E1 -5999.889,E2 -5999.889} C_VEL
LIN {X 0,Y 495.815,Z 207.721,A -85,B 0,C 180,E1 -6000.565,E2 -6000.565} C_VEL
LIN {X 0,Y 495.738,Z 207.729,A -85,B 0,C 180,E1 -6000.794,E2 -6000.794} C_VEL
LIN {X 0,Y 495.769,Z 207.734,A -85,B 0,C 180,E1 -6003.935,E2 -6003.935} C_VEL
LIN {X 0,Y 495.75,Z 207.728,A -85,B 0,C 180,E1 -6007.143,E2 -6007.143} C_VEL
LIN {X 0,Y 495.761,Z 207.73,A -85,B 0,C 180,E1 -6010.113,E2 -6010.113} C_VEL
LIN {X 0,Y 495.75,Z 207.727,A -85,B 0,C 180,E1 -6012.683,E2 -6012.683} C_VEL
LIN {X 0,Y 495.779,Z 207.726,A -85,B 0,C 180,E1 -6015.22,E2 -6015.22} C_VEL
LIN {X 0,Y 495.85,Z 207.718,A -85,B 0,C 180,E1 -6018.557,E2 -6018.557} C_VEL
LIN {X 0,Y 495.877,Z 207.845,A -85,B 0,C 180,E1 -6021.675,E2 -6021.675} C_VEL
LIN {X 0,Y 496.517,Z 213.856,A -85,B 0,C 180,E1 -6022.888,E2 -6022.888} C_VEL
LIN {X 0,Y 496.201,Z 224.852,A -85,B 0,C 180,E1 -6025.025,E2 -6025.025} C_VEL
LIN {X 0,Y 498.679,Z 237.589,A -85,B 0,C 180,E1 -6025.303,E2 -6025.303} C_VEL
LIN {X 0,Y 497.972,Z 332.158,A -85,B 0,C 180,E1 -6026.69,E2 -6026.69} C_VEL
LIN {X 0,Y 497.771,Z 345.832,A -85,B 0,C 180,E1 -6027.068,E2 -6027.068} C_VEL
LIN {X 0,Y 497.512,Z 358.125,A -85,B 0,C 180,E1 -6027.573,E2 -6027.573} C_VEL
LIN {X 0,Y 497.234,Z 369.123,A -85,B 0,C 180,E1 -6028.179,E2 -6028.179} C_VEL
LIN {X 0,Y 496.752,Z 380.597,A -85,B 0,C 180,E1 -6028.988,E2 -6028.988} C_VEL
LIN {X 0,Y 496.42,Z 390.895,A -85,B 0,C 180,E1 -6029.9,E2 -6029.9} C_VEL
LIN {X 0,Y 496.133,Z 399.338,A -85,B 0,C 180,E1 -6030.813,E2 -6030.813} C_VEL
LIN {X 0,Y 495.789,Z 407.152,A -85,B 0,C 180,E1 -6031.829,E2 -6031.829} C_VEL
LIN {X 0,Y 495.53,Z 414.807,A -85,B 0,C 180,E1 -6033.05,E2 -6033.05} C_VEL
LIN {X 0,Y 495.371,Z 421.842,A -85,B 0,C 180,E1 -6034.476,E2 -6034.476} C_VEL
LIN {X 0,Y 495.214,Z 426.558,A -85,B 0,C 180,E1 -6035.702,E2 -6035.702} C_VEL
LIN {X 0,Y 495.14,Z 430.177,A -85,B 0,C 180,E1 -6036.93,E2 -6036.93} C_VEL
LIN {X 0,Y 495.018,Z 432.799,A -85,B 0,C 180,E1 -6038.163,E2 -6038.163} C_VEL
LIN {X 0,Y 494.998,Z 434.032,A -85,B 0,C 180,E1 -6038.986,E2 -6038.986} C_VEL
LIN {X 0,Y 494.961,Z 434.845,A -85,B 0,C 180,E1 -6039.811,E2 -6039.811} C_VEL
LIN {X 0,Y 494.998,Z 435.231,A -85,B 0,C 180,E1 -6040.637,E2 -6040.637} C_VEL
LIN {X 0,Y 495.01,Z 435.209,A -85,B 0,C 180,E1 -6041.58,E2 -6041.58} C_VEL
LIN {X 0,Y 494.969,Z 434.01,A -85,B 0,C 180,E1 -6043.131,E2 -6043.131} C_VEL
LIN {X 0,Y 495.016,Z 432.749,A -85,B 0,C 180,E1 -6043.967,E2 -6043.967} C_VEL
LIN {X 0,Y 495.119,Z 430.23,A -85,B 0,C 180,E1 -6045.152,E2 -6045.152} C_VEL
LIN {X 0,Y 495.215,Z 426.254,A -85,B 0,C 180,E1 -6046.489,E2 -6046.489} C_VEL
LIN {X 0,Y 495.355,Z 421.394,A -85,B 0,C 180,E1 -6047.73,E2 -6047.73} C_VEL
LIN {X 0,Y 495.543,Z 414.892,A -85,B 0,C 180,E1 -6049.038,E2 -6049.038} C_VEL
LIN {X 0,Y 495.914,Z 406.832,A -85,B 0,C 180,E1 -6050.316,E2 -6050.316} C_VEL
LIN {X 0,Y 496.202,Z 398.485,A -85,B 0,C 180,E1 -6051.389,E2 -6051.389} C_VEL
LIN {X 0,Y 496.587,Z 388.198,A -85,B 0,C 180,E1 -6052.464,E2 -6052.464} C_VEL
LIN {X 0,Y 496.966,Z 377.907,A -85,B 0,C 180,E1 -6053.326,E2 -6053.326} C_VEL
LIN {X 0,Y 497.314,Z 366.541,A -85,B 0,C 180,E1 -6054.082,E2 -6054.082} C_VEL
LIN {X 0,Y 497.641,Z 353.822,A -85,B 0,C 180,E1 -6054.732,E2 -6054.732} C_VEL
LIN {X 0,Y 497.916,Z 340.856,A -85,B 0,C 180,E1 -6055.199,E2 -6055.199} C_VEL
LIN {X 0,Y 498.068,Z 327.528,A -85,B 0,C 180,E1 -6055.502,E2 -6055.502} C_VEL
LIN {X 0,Y 498.597,Z 236.174,A -85,B 0,C 180,E1 -6056.836,E2 -6056.836} C_VEL
LIN {X 0,Y 496.346,Z 224.83,A -85,B 0,C 180,E1 -6057.105,E2 -6057.105} C_VEL
LIN {X 0,Y 496.405,Z 211.415,A -85,B 0,C 180,E1 -6059.703,E2 -6059.703} C_VEL
LIN {X 0,Y 495.792,Z 207.73,A -85,B 0,C 180,E1 -6060.466,E2 -6060.466} C_VEL
LIN {X 0,Y 495.756,Z 207.729,A -85,B 0,C 180,E1 -6063.563,E2 -6063.563} C_VEL
LIN {X 0,Y 495.727,Z 207.738,A -85,B 0,C 180,E1 -6066.542,E2 -6066.542} C_VEL
LIN {X 0,Y 495.774,Z 207.729,A -85,B 0,C 180,E1 -6069.634,E2 -6069.634} C_VEL
LIN {X 0,Y 495.726,Z 207.737,A -85,B 0,C 180,E1 -6072.505,E2 -6072.505} C_VEL
LIN {X 0,Y 495.736,Z 207.73,A -85,B 0,C 180,E1 -6075.138,E2 -6075.138} C_VEL
LIN {X 0,Y 495.764,Z 207.734,A -85,B 0,C 180,E1 -6078.219,E2 -6078.219} C_VEL
LIN {X 0,Y 495.75,Z 207.729,A -85,B 0,C 180,E1 -6081.229,E2 -6081.229} C_VEL
LIN {X 0,Y 495.737,Z 207.732,A -85,B 0,C 180,E1 -6084.461,E2 -6084.461} C_VEL
LIN {X 0,Y 495.747,Z 207.731,A -85,B 0,C 180,E1 -6087.404,E2 -6087.404} C_VEL
LIN {X 0,Y 495.758,Z 207.73,A -85,B 0,C 180,E1 -6090.253,E2 -6090.253} C_VEL
LIN {X 0,Y 495.798,Z 207.721,A -85,B 0,C 180,E1 -6093.249,E2 -6093.249} C_VEL
LIN {X 0,Y 495.732,Z 207.735,A -85,B 0,C 180,E1 -6095.724,E2 -6095.724} C_VEL
LIN {X 0,Y 495.731,Z 207.731,A -85,B 0,C 180,E1 -6098.37,E2 -6098.37} C_VEL
LIN {X 0,Y 495.756,Z 207.725,A -85,B 0,C 180,E1 -6100.97,E2 -6100.97} C_VEL
LIN {X 0,Y 495.758,Z 207.733,A -85,B 0,C 180,E1 -6103.529,E2 -6103.529} C_VEL
LIN {X 0,Y 495.762,Z 207.728,A -85,B 0,C 180,E1 -6106.055,E2 -6106.055} C_VEL
LIN {X 0,Y 495.821,Z 207.717,A -85,B 0,C 180,E1 -6108.554,E2 -6108.554} C_VEL
LIN {X 0,Y 495.843,Z 207.718,A -85,B 0,C 180,E1 -6111.851,E2 -6111.851} C_VEL
LIN {X 0,Y 495.873,Z 207.71,A -85,B 0,C 180,E1 -6114.306,E2 -6114.306} C_VEL
LIN {X 0,Y 495.956,Z 207.703,A -85,B 0,C 180,E1 -6117.563,E2 -6117.563} C_VEL
LIN {X 0,Y 495.957,Z 207.702,A -85,B 0,C 180,E1 -6120,E2 -6120} C_VEL
LIN {X 0,Y 495.955,Z 207.701,A -85,B 0,C 180,E1 -6122.436,E2 -6122.436} C_VEL
LIN {X 0,Y 495.852,Z 207.716,A -85,B 0,C 180,E1 -6125.694,E2 -6125.694} C_VEL
LIN {X 0,Y 495.802,Z 207.718,A -85,B 0,C 180,E1 -6128.149,E2 -6128.149} C_VEL
LIN {X 0,Y 495.838,Z 207.716,A -85,B 0,C 180,E1 -6131.445,E2 -6131.445} C_VEL
LIN {X 0,Y 495.754,Z 207.734,A -85,B 0,C 180,E1 -6134.784,E2 -6134.784} C_VEL
LIN {X 0,Y 495.73,Z 207.731,A -85,B 0,C 180,E1 -6137.321,E2 -6137.321} C_VEL
LIN {X 0,Y 495.738,Z 207.729,A -85,B 0,C 180,E1 -6139.892,E2 -6139.892} C_VEL
LIN {X 0,Y 495.728,Z 207.737,A -85,B 0,C 180,E1 -6142.861,E2 -6142.861} C_VEL
LIN {X 0,Y 495.729,Z 207.729,A -85,B 0,C 180,E1 -6146.071,E2 -6146.071} C_VEL
LIN {X 0,Y 495.719,Z 207.735,A -85,B 0,C 180,E1 -6148.818,E2 -6148.818} C_VEL
LIN {X 0,Y 495.729,Z 207.731,A -85,B 0,C 180,E1 -6151.726,E2 -6151.726} C_VEL
LIN {X 0,Y 495.738,Z 207.735,A -85,B 0,C 180,E1 -6154.694,E2 -6154.694} C_VEL
LIN {X 0,Y 495.707,Z 207.729,A -85,B 0,C 180,E1 -6157.564,E2 -6157.564} C_VEL
LIN {X 0,Y 495.747,Z 207.732,A -85,B 0,C 180,E1 -6160.702,E2 -6160.702} C_VEL
LIN {X 0,Y 495.712,Z 207.737,A -85,B 0,C 180,E1 -6164.004,E2 -6164.004} C_VEL
LIN {X 0,Y 495.703,Z 207.734,A -85,B 0,C 180,E1 -6167.118,E2 -6167.118} C_VEL
LIN {X 0,Y 495.733,Z 207.735,A -85,B 0,C 180,E1 -6170.362,E2 -6170.362} C_VEL
LIN {X 0,Y 495.72,Z 207.735,A -85,B 0,C 180,E1 -6173.458,E2 -6173.458} C_VEL
LIN {X 0,Y 495.753,Z 207.73,A -85,B 0,C 180,E1 -6176.437,E2 -6176.437} C_VEL
LIN {X 0,Y 495.747,Z 207.732,A -85,B 0,C 180,E1 -6179.314,E2 -6179.314} C_VEL
LIN {X 0,Y 495.738,Z 207.735,A -85,B 0,C 180,E1 -6182.107,E2 -6182.107} C_VEL
LIN {X 0,Y 495.824,Z 207.826,A -85,B 0,C 180,E1 -6184.302,E2 -6184.302} C_VEL
LIN {X 0,Y 497.678,Z 217.824,A -85,B 0,C 180,E1 -6186.048,E2 -6186.048} C_VEL
LIN {X 0,Y 497.279,Z 232.655,A -85,B 0,C 180,E1 -6188.442,E2 -6188.442} C_VEL
LIN {X 0,Y 496.582,Z 254.219,A -85,B 0,C 180,E1 -6191.859,E2 -6191.859} C_VEL
LIN {X 0,Y 496.227,Z 267.755,A -85,B 0,C 180,E1 -6193.95,E2 -6193.95} C_VEL
LIN {X 0,Y 498.477,Z 284.174,A -85,B 0,C 180,E1 -6194.268,E2 -6194.268} C_VEL
LIN {X 0,Y 497.955,Z 376.19,A -85,B 0,C 180,E1 -6195.622,E2 -6195.622} C_VEL
LIN {X 0,Y 497.667,Z 389.464,A -85,B 0,C 180,E1 -6195.979,E2 -6195.979} C_VEL
LIN {X 0,Y 497.218,Z 402.762,A -85,B 0,C 180,E1 -6196.513,E2 -6196.513} C_VEL
LIN {X 0,Y 496.922,Z 413.974,A -85,B 0,C 180,E1 -6197.131,E2 -6197.131} C_VEL
LIN {X 0,Y 496.473,Z 425.563,A -85,B 0,C 180,E1 -6197.948,E2 -6197.948} C_VEL
LIN {X 0,Y 496.122,Z 436.045,A -85,B 0,C 180,E1 -6198.871,E2 -6198.871} C_VEL
LIN {X 0,Y 495.809,Z 444.619,A -85,B 0,C 180,E1 -6199.794,E2 -6199.794} C_VEL
LIN {X 0,Y 495.541,Z 452.535,A -85,B 0,C 180,E1 -6200.818,E2 -6200.818} C_VEL
LIN {X 0,Y 495.322,Z 460.272,A -85,B 0,C 180,E1 -6202.047,E2 -6202.047} C_VEL
LIN {X 0,Y 495.165,Z 467.408,A -85,B 0,C 180,E1 -6203.479,E2 -6203.479} C_VEL
LIN {X 0,Y 495.102,Z 472.16,A -85,B 0,C 180,E1 -6204.705,E2 -6204.705} C_VEL
LIN {X 0,Y 495.035,Z 475.79,A -85,B 0,C 180,E1 -6205.928,E2 -6205.928} C_VEL
LIN {X 0,Y 495.042,Z 477.666,A -85,B 0,C 180,E1 -6206.743,E2 -6206.743} C_VEL
LIN {X 0,Y 495.025,Z 479.072,A -85,B 0,C 180,E1 -6207.558,E2 -6207.558} C_VEL
LIN {X 0,Y 494.916,Z 480.687,A -85,B 0,C 180,E1 -6209.185,E2 -6209.185} C_VEL
LIN {X 0,Y 494.909,Z 480.907,A -85,B 0,C 180,E1 -6209.998,E2 -6209.998} C_VEL
LIN {X 0,Y 494.963,Z 480.09,A -85,B 0,C 180,E1 -6211.626,E2 -6211.626} C_VEL
LIN {X 0,Y 495.024,Z 479.096,A -85,B 0,C 180,E1 -6212.439,E2 -6212.439} C_VEL
LIN {X 0,Y 495.041,Z 477.697,A -85,B 0,C 180,E1 -6213.254,E2 -6213.254} C_VEL
LIN {X 0,Y 495.007,Z 474.75,A -85,B 0,C 180,E1 -6214.477,E2 -6214.477} C_VEL
LIN {X 0,Y 495.115,Z 470.766,A -85,B 0,C 180,E1 -6215.7,E2 -6215.7} C_VEL
LIN {X 0,Y 495.237,Z 464.634,A -85,B 0,C 180,E1 -6217.131,E2 -6217.131} C_VEL
LIN {X 0,Y 495.412,Z 457.935,A -85,B 0,C 180,E1 -6218.359,E2 -6218.359} C_VEL
LIN {X 0,Y 495.656,Z 449.623,A -85,B 0,C 180,E1 -6219.588,E2 -6219.588} C_VEL
LIN {X 0,Y 495.965,Z 441.104,A -85,B 0,C 180,E1 -6220.613,E2 -6220.613} C_VEL
LIN {X 0,Y 496.387,Z 430.582,A -85,B 0,C 180,E1 -6221.637,E2 -6221.637} C_VEL
LIN {X 0,Y 496.737,Z 418.732,A -85,B 0,C 180,E1 -6222.561,E2 -6222.561} C_VEL
LIN {X 0,Y 497.131,Z 406.822,A -85,B 0,C 180,E1 -6223.278,E2 -6223.278} C_VEL
LIN {X 0,Y 497.484,Z 394.43,A -85,B 0,C 180,E1 -6223.841,E2 -6223.841} C_VEL
LIN {X 0,Y 497.813,Z 381.686,A -85,B 0,C 180,E1 -6224.248,E2 -6224.248} C_VEL
LIN {X 0,Y 498.053,Z 368.286,A -85,B 0,C 180,E1 -6224.502,E2 -6224.502} C_VEL
LIN {X 0,Y 498.438,Z 283.104,A -85,B 0,C 180,E1 -6225.736,E2 -6225.736} C_VEL
LIN {X 0,Y 496.228,Z 267.699,A -85,B 0,C 180,E1 -6226.034,E2 -6226.034} C_VEL
LIN {X 0,Y 496.728,Z 248.807,A -85,B 0,C 180,E1 -6228.987,E2 -6228.987} C_VEL
LIN {X 0,Y 497.293,Z 229.796,A -85,B 0,C 180,E1 -6231.99,E2 -6231.99} C_VEL
LIN {X 0,Y 497.619,Z 217.518,A -85,B 0,C 180,E1 -6233.952,E2 -6233.952} C_VEL
LIN {X 0,Y 495.821,Z 207.726,A -85,B 0,C 180,E1 -6235.639,E2 -6235.639} C_VEL
LIN {X 0,Y 495.756,Z 207.73,A -85,B 0,C 180,E1 -6238.811,E2 -6238.811} C_VEL
LIN {X 0,Y 495.737,Z 207.735,A -85,B 0,C 180,E1 -6241.721,E2 -6241.721} C_VEL
LIN {X 0,Y 495.755,Z 207.728,A -85,B 0,C 180,E1 -6244.691,E2 -6244.691} C_VEL
LIN {X 0,Y 495.706,Z 207.736,A -85,B 0,C 180,E1 -6247.557,E2 -6247.557} C_VEL
LIN {X 0,Y 495.739,Z 207.729,A -85,B 0,C 180,E1 -6250.696,E2 -6250.696} C_VEL
LIN {X 0,Y 495.702,Z 207.74,A -85,B 0,C 180,E1 -6253.997,E2 -6253.997} C_VEL
LIN {X 0,Y 495.729,Z 207.731,A -85,B 0,C 180,E1 -6257.117,E2 -6257.117} C_VEL
LIN {X 0,Y 495.757,Z 207.728,A -85,B 0,C 180,E1 -6260.362,E2 -6260.362} C_VEL
LIN {X 0,Y 495.693,Z 207.74,A -85,B 0,C 180,E1 -6263.453,E2 -6263.453} C_VEL
LIN {X 0,Y 495.718,Z 207.732,A -85,B 0,C 180,E1 -6266.432,E2 -6266.432} C_VEL
LIN {X 0,Y 495.713,Z 207.737,A -85,B 0,C 180,E1 -6269.31,E2 -6269.31} C_VEL
LIN {X 0,Y 495.735,Z 207.731,A -85,B 0,C 180,E1 -6272.106,E2 -6272.106} C_VEL
LIN {X 0,Y 495.742,Z 207.729,A -85,B 0,C 180,E1 -6274.83,E2 -6274.83} C_VEL
LIN {X 0,Y 495.734,Z 207.737,A -85,B 0,C 180,E1 -6277.494,E2 -6277.494} C_VEL
LIN {X 0,Y 495.734,Z 207.73,A -85,B 0,C 180,E1 -6280.108,E2 -6280.108} C_VEL
LIN {X 0,Y 495.74,Z 207.729,A -85,B 0,C 180,E1 -6282.68,E2 -6282.68} C_VEL
LIN {X 0,Y 495.738,Z 207.736,A -85,B 0,C 180,E1 -6285.216,E2 -6285.216} C_VEL
LIN {X 0,Y 495.822,Z 207.719,A -85,B 0,C 180,E1 -6288.554,E2 -6288.554} C_VEL
LIN {X 0,Y 495.828,Z 207.719,A -85,B 0,C 180,E1 -6291.851,E2 -6291.851} C_VEL
LIN {X 0,Y 495.861,Z 207.714,A -85,B 0,C 180,E1 -6294.306,E2 -6294.306} C_VEL
LIN {X 0,Y 495.937,Z 207.706,A -85,B 0,C 180,E1 -6297.563,E2 -6297.563} C_VEL
LIN {X 0,Y 495.933,Z 207.704,A -85,B 0,C 180,E1 -6300,E2 -6300} C_VEL
LIN {X 0,Y 495.932,Z 207.706,A -85,B 0,C 180,E1 -6302.437,E2 -6302.437} C_VEL
LIN {X 0,Y 495.843,Z 207.716,A -85,B 0,C 180,E1 -6305.694,E2 -6305.694} C_VEL
LIN {X 0,Y 495.814,Z 207.72,A -85,B 0,C 180,E1 -6308.149,E2 -6308.149} C_VEL
LIN {X 0,Y 495.816,Z 207.72,A -85,B 0,C 180,E1 -6311.446,E2 -6311.446} C_VEL
LIN {X 0,Y 495.738,Z 207.738,A -85,B 0,C 180,E1 -6314.785,E2 -6314.785} C_VEL
LIN {X 0,Y 495.74,Z 207.73,A -85,B 0,C 180,E1 -6317.32,E2 -6317.32} C_VEL
LIN {X 0,Y 495.718,Z 207.732,A -85,B 0,C 180,E1 -6319.893,E2 -6319.893} C_VEL
LIN {X 0,Y 495.713,Z 207.737,A -85,B 0,C 180,E1 -6322.865,E2 -6322.865} C_VEL
LIN {X 0,Y 495.749,Z 207.729,A -85,B 0,C 180,E1 -6326.07,E2 -6326.07} C_VEL
LIN {X 0,Y 495.735,Z 207.734,A -85,B 0,C 180,E1 -6328.817,E2 -6328.817} C_VEL
LIN {X 0,Y 495.714,Z 207.732,A -85,B 0,C 180,E1 -6331.729,E2 -6331.729} C_VEL
LIN {X 0,Y 495.734,Z 207.734,A -85,B 0,C 180,E1 -6334.699,E2 -6334.699} C_VEL
LIN {X 0,Y 495.691,Z 207.735,A -85,B 0,C 180,E1 -6337.565,E2 -6337.565} C_VEL
LIN {X 0,Y 495.742,Z 207.732,A -85,B 0,C 180,E1 -6340.703,E2 -6340.703} C_VEL
LIN {X 0,Y 495.701,Z 207.735,A -85,B 0,C 180,E1 -6343.699,E2 -6343.699} C_VEL
LIN {X 0,Y 495.698,Z 207.741,A -85,B 0,C 180,E1 -6346.31,E2 -6346.31} C_VEL
LIN {X 0,Y 495.74,Z 207.729,A -85,B 0,C 180,E1 -6349.304,E2 -6349.304} C_VEL
LIN {X 0,Y 495.707,Z 207.737,A -85,B 0,C 180,E1 -6352.443,E2 -6352.443} C_VEL
LIN {X 0,Y 495.763,Z 207.727,A -85,B 0,C 180,E1 -6355.461,E2 -6355.461} C_VEL
LIN {X 0,Y 495.737,Z 207.733,A -85,B 0,C 180,E1 -6358.368,E2 -6358.368} C_VEL
LIN {X 0,Y 495.738,Z 207.729,A -85,B 0,C 180,E1 -6360.794,E2 -6360.794} C_VEL
LIN {X 0,Y 495.083,Z 207.814,A -85,B 0,C 180,E1 -6361.473,E2 -6361.473} C_VEL
LIN {X 0,Y 492.225,Z 208.168,A -85,B 0,C 180,E1 -6362.575,E2 -6362.575} C_VEL
LIN {X 0,Y 489.811,Z 208.47,A -85,B 0,C 180,E1 -6363.464,E2 -6363.464} C_VEL
LIN {X 0,Y 488.788,Z 208.6,A -85,B 0,C 180,E1 -6364.15,E2 -6364.15} C_VEL
LIN {X 0,Y 488.713,Z 208.605,A -85,B 0,C 180,E1 -6364.383,E2 -6364.383} C_VEL
LIN {X 0,Y 488.712,Z 208.605,A -85,B 0,C 180,E1 -6367.157,E2 -6367.157} C_VEL
LIN {X 0,Y 488.716,Z 208.612,A -85,B 0,C 180,E1 -6369.814,E2 -6369.814} C_VEL
LIN {X 0,Y 488.703,Z 208.606,A -85,B 0,C 180,E1 -6372.426,E2 -6372.426} C_VEL
LIN {X 0,Y 488.754,Z 208.6,A -85,B 0,C 180,E1 -6375.002,E2 -6375.002} C_VEL
LIN {X 0,Y 488.804,Z 208.596,A -85,B 0,C 180,E1 -6378.39,E2 -6378.39} C_VEL
LIN {X 0,Y 488.831,Z 208.616,A -85,B 0,C 180,E1 -6381.528,E2 -6381.528} C_VEL
LIN {X 0,Y 489.541,Z 214.802,A -85,B 0,C 180,E1 -6382.786,E2 -6382.786} C_VEL
LIN {X 0,Y 489.296,Z 225.088,A -85,B 0,C 180,E1 -6384.8,E2 -6384.8} C_VEL
LIN {X 0,Y 491.778,Z 237.564,A -85,B 0,C 180,E1 -6385.083,E2 -6385.083} C_VEL
LIN {X 0,Y 491.087,Z 332.243,A -85,B 0,C 180,E1 -6386.489,E2 -6386.489} C_VEL
LIN {X 0,Y 490.887,Z 345.255,A -85,B 0,C 180,E1 -6386.847,E2 -6386.847} C_VEL
LIN {X 0,Y 490.607,Z 358.342,A -85,B 0,C 180,E1 -6387.385,E2 -6387.385} C_VEL
LIN {X 0,Y 490.285,Z 370.155,A -85,B 0,C 180,E1 -6388.051,E2 -6388.051} C_VEL
LIN {X 0,Y 489.788,Z 381.504,A -85,B 0,C 180,E1 -6388.871,E2 -6388.871} C_VEL
LIN {X 0,Y 489.431,Z 391.711,A -85,B 0,C 180,E1 -6389.796,E2 -6389.796} C_VEL
LIN {X 0,Y 489.088,Z 400.921,A -85,B 0,C 180,E1 -6390.825,E2 -6390.825} C_VEL
LIN {X 0,Y 488.685,Z 409.851,A -85,B 0,C 180,E1 -6392.062,E2 -6392.062} C_VEL
LIN {X 0,Y 488.417,Z 417.059,A -85,B 0,C 180,E1 -6393.301,E2 -6393.301} C_VEL
LIN {X 0,Y 488.29,Z 422.839,A -85,B 0,C 180,E1 -6394.542,E2 -6394.542} C_VEL
LIN {X 0,Y 488.147,Z 427.413,A -85,B 0,C 180,E1 -6395.785,E2 -6395.785} C_VEL
LIN {X 0,Y 488.096,Z 429.838,A -85,B 0,C 180,E1 -6396.616,E2 -6396.616} C_VEL
LIN {X 0,Y 488.003,Z 431.824,A -85,B 0,C 180,E1 -6397.448,E2 -6397.448} C_VEL
LIN {X 0,Y 487.937,Z 433.398,A -85,B 0,C 180,E1 -6398.282,E2 -6398.282} C_VEL
LIN {X 0,Y 487.914,Z 434.546,A -85,B 0,C 180,E1 -6399.117,E2 -6399.117} C_VEL
LIN {X 0,Y 487.904,Z 435.589,A -85,B 0,C 180,E1 -6400.793,E2 -6400.793} C_VEL
LIN {X 0,Y 487.931,Z 435.528,A -85,B 0,C 180,E1 -6401.634,E2 -6401.634} C_VEL
LIN {X 0,Y 487.881,Z 435.041,A -85,B 0,C 180,E1 -6402.479,E2 -6402.479} C_VEL
LIN {X 0,Y 487.893,Z 434.123,A -85,B 0,C 180,E1 -6403.325,E2 -6403.325} C_VEL
LIN {X 0,Y 487.943,Z 432.799,A -85,B 0,C 180,E1 -6404.174,E2 -6404.174} C_VEL
LIN {X 0,Y 488.055,Z 430.48,A -85,B 0,C 180,E1 -6405.246,E2 -6405.246} C_VEL
LIN {X 0,Y 488.173,Z 426.036,A -85,B 0,C 180,E1 -6406.734,E2 -6406.734} C_VEL
LIN {X 0,Y 488.326,Z 421.355,A -85,B 0,C 180,E1 -6407.917,E2 -6407.917} C_VEL
LIN {X 0,Y 488.504,Z 415.515,A -85,B 0,C 180,E1 -6409.105,E2 -6409.105} C_VEL
LIN {X 0,Y 488.889,Z 407.761,A -85,B 0,C 180,E1 -6410.373,E2 -6410.373} C_VEL
LIN {X 0,Y 489.221,Z 399.304,A -85,B 0,C 180,E1 -6411.489,E2 -6411.489} C_VEL
LIN {X 0,Y 489.621,Z 389.124,A -85,B 0,C 180,E1 -6412.579,E2 -6412.579} C_VEL
LIN {X 0,Y 490.041,Z 378.936,A -85,B 0,C 180,E1 -6413.458,E2 -6413.458} C_VEL
LIN {X 0,Y 490.424,Z 367.894,A -85,B 0,C 180,E1 -6414.217,E2 -6414.217} C_VEL
LIN {X 0,Y 490.741,Z 355.467,A -85,B 0,C 180,E1 -6414.877,E2 -6414.877} C_VEL
LIN {X 0,Y 491.054,Z 342.64,A -85,B 0,C 180,E1 -6415.369,E2 -6415.369} C_VEL
LIN {X 0,Y 491.251,Z 329.603,A -85,B 0,C 180,E1 -6415.687,E2 -6415.687} C_VEL
LIN {X 0,Y 491.85,Z 237.212,A -85,B 0,C 180,E1 -6417.061,E2 -6417.061} C_VEL
LIN {X 0,Y 489.393,Z 225.114,A -85,B 0,C 180,E1 -6417.356,E2 -6417.356} C_VEL
LIN {X 0,Y 489.487,Z 213.158,A -85,B 0,C 180,E1 -6419.691,E2 -6419.691} C_VEL
LIN {X 0,Y 488.731,Z 208.609,A -85,B 0,C 180,E1 -6420.636,E2 -6420.636} C_VEL
LIN {X 0,Y 488.73,Z 208.608,A -85,B 0,C 180,E1 -6424.111,E2 -6424.111} C_VEL
LIN {X 0,Y 488.676,Z 208.613,A -85,B 0,C 180,E1 -6427.157,E2 -6427.157} C_VEL
LIN {X 0,Y 488.734,Z 208.606,A -85,B 0,C 180,E1 -6429.249,E2 -6429.249} C_VEL
LIN {X 0,Y 488.701,Z 208.61,A -85,B 0,C 180,E1 -6431.599,E2 -6431.599} C_VEL
LIN {X 0,Y 488.699,Z 208.608,A -85,B 0,C 180,E1 -6434.8,E2 -6434.8} C_VEL
LIN {X 0,Y 488.721,Z 208.606,A -85,B 0,C 180,E1 -6437.477,E2 -6437.477} C_VEL
LIN {X 0,Y 488.725,Z 208.605,A -85,B 0,C 180,E1 -6440.748,E2 -6440.748} C_VEL
LIN {X 0,Y 488.665,Z 208.616,A -85,B 0,C 180,E1 -6443.867,E2 -6443.867} C_VEL
LIN {X 0,Y 488.718,Z 208.604,A -85,B 0,C 180,E1 -6446.875,E2 -6446.875} C_VEL
LIN {X 0,Y 488.71,Z 208.61,A -85,B 0,C 180,E1 -6449.78,E2 -6449.78} C_VEL
LIN {X 0,Y 488.767,Z 208.596,A -85,B 0,C 180,E1 -6453.055,E2 -6453.055} C_VEL
LIN {X 0,Y 488.673,Z 208.609,A -85,B 0,C 180,E1 -6456.253,E2 -6456.253} C_VEL
LIN {X 0,Y 488.719,Z 208.606,A -85,B 0,C 180,E1 -6459.174,E2 -6459.174} C_VEL
LIN {X 0,Y 488.71,Z 208.605,A -85,B 0,C 180,E1 -6462.422,E2 -6462.422} C_VEL
LIN {X 0,Y 488.73,Z 208.601,A -85,B 0,C 180,E1 -6464.998,E2 -6464.998} C_VEL
LIN {X 0,Y 488.775,Z 208.595,A -85,B 0,C 180,E1 -6468.387,E2 -6468.387} C_VEL
LIN {X 0,Y 488.787,Z 208.598,A -85,B 0,C 180,E1 -6471.733,E2 -6471.733} C_VEL
LIN {X 0,Y 488.833,Z 208.588,A -85,B 0,C 180,E1 -6474.224,E2 -6474.224} C_VEL
LIN {X 0,Y 488.925,Z 208.579,A -85,B 0,C 180,E1 -6477.528,E2 -6477.528} C_VEL
LIN {X 0,Y 488.929,Z 208.578,A -85,B 0,C 180,E1 -6480,E2 -6480} C_VEL
LIN {X 0,Y 488.923,Z 208.577,A -85,B 0,C 180,E1 -6482.471,E2 -6482.471} C_VEL
LIN {X 0,Y 488.81,Z 208.593,A -85,B 0,C 180,E1 -6485.776,E2 -6485.776} C_VEL
LIN {X 0,Y 488.751,Z 208.596,A -85,B 0,C 180,E1 -6488.267,E2 -6488.267} C_VEL
LIN {X 0,Y 488.794,Z 208.592,A -85,B 0,C 180,E1 -6491.613,E2 -6491.613} C_VEL
LIN {X 0,Y 488.728,Z 208.608,A -85,B 0,C 180,E1 -6495.001,E2 -6495.001} C_VEL
LIN {X 0,Y 488.716,Z 208.606,A -85,B 0,C 180,E1 -6498.444,E2 -6498.444} C_VEL
LIN {X 0,Y 488.677,Z 208.61,A -85,B 0,C 180,E1 -6501.072,E2 -6501.072} C_VEL
LIN {X 0,Y 488.643,Z 208.613,A -85,B 0,C 180,E1 -6503.748,E2 -6503.748} C_VEL
LIN {X 0,Y 488.698,Z 208.611,A -85,B 0,C 180,E1 -6506.929,E2 -6506.929} C_VEL
LIN {X 0,Y 488.697,Z 208.608,A -85,B 0,C 180,E1 -6510.221,E2 -6510.221} C_VEL
LIN {X 0,Y 488.687,Z 208.605,A -85,B 0,C 180,E1 -6513.481,E2 -6513.481} C_VEL
LIN {X 0,Y 488.66,Z 208.617,A -85,B 0,C 180,E1 -6516.356,E2 -6516.356} C_VEL
LIN {X 0,Y 488.676,Z 208.604,A -85,B 0,C 180,E1 -6519.257,E2 -6519.257} C_VEL
LIN {X 0,Y 488.69,Z 208.609,A -85,B 0,C 180,E1 -6521.601,E2 -6521.601} C_VEL
LIN {X 0,Y 488.686,Z 208.609,A -85,B 0,C 180,E1 -6524.805,E2 -6524.805} C_VEL
LIN {X 0,Y 488.675,Z 208.61,A -85,B 0,C 180,E1 -6527.476,E2 -6527.476} C_VEL
LIN {X 0,Y 488.683,Z 208.609,A -85,B 0,C 180,E1 -6530.747,E2 -6530.747} C_VEL
LIN {X 0,Y 488.671,Z 208.618,A -85,B 0,C 180,E1 -6533.87,E2 -6533.87} C_VEL
LIN {X 0,Y 488.732,Z 208.602,A -85,B 0,C 180,E1 -6536.879,E2 -6536.879} C_VEL
LIN {X 0,Y 488.719,Z 208.611,A -85,B 0,C 180,E1 -6539.782,E2 -6539.782} C_VEL
LIN {X 0,Y 488.723,Z 208.607,A -85,B 0,C 180,E1 -6543.073,E2 -6543.073} C_VEL
LIN {X 0,Y 488.752,Z 208.66,A -85,B 0,C 180,E1 -6544.074,E2 -6544.074} C_VEL
LIN {X 0,Y 490.751,Z 218.98,A -85,B 0,C 180,E1 -6545.912,E2 -6545.912} C_VEL
LIN {X 0,Y 490.465,Z 229.751,A -85,B 0,C 180,E1 -6547.684,E2 -6547.684} C_VEL
LIN {X 0,Y 489.76,Z 250.829,A -85,B 0,C 180,E1 -6551.089,E2 -6551.089} C_VEL
LIN {X 0,Y 489.238,Z 267.163,A -85,B 0,C 180,E1 -6553.69,E2 -6553.69} C_VEL
LIN {X 0,Y 491.68,Z 284.554,A -85,B 0,C 180,E1 -6554.045,E2 -6554.045} C_VEL
LIN {X 0,Y 491.103,Z 376.244,A -85,B 0,C 180,E1 -6555.417,E2 -6555.417} C_VEL
LIN {X 0,Y 490.762,Z 390.14,A -85,B 0,C 180,E1 -6555.804,E2 -6555.804} C_VEL
LIN {X 0,Y 490.322,Z 402.592,A -85,B 0,C 180,E1 -6556.32,E2 -6556.32} C_VEL
LIN {X 0,Y 489.963,Z 414.031,A -85,B 0,C 180,E1 -6556.964,E2 -6556.964} C_VEL
LIN {X 0,Y 489.514,Z 425.307,A -85,B 0,C 180,E1 -6557.774,E2 -6557.774} C_VEL
LIN {X 0,Y 489.129,Z 435.764,A -85,B 0,C 180,E1 -6558.71,E2 -6558.71} C_VEL
LIN {X 0,Y 488.783,Z 444.322,A -85,B 0,C 180,E1 -6559.645,E2 -6559.645} C_VEL
LIN {X 0,Y 488.481,Z 452.225,A -85,B 0,C 180,E1 -6560.685,E2 -6560.685} C_VEL
LIN {X 0,Y 488.251,Z 459.952,A -85,B 0,C 180,E1 -6561.931,E2 -6561.931} C_VEL
LIN {X 0,Y 488.074,Z 467.082,A -85,B 0,C 180,E1 -6563.384,E2 -6563.384} C_VEL
LIN {X 0,Y 488.013,Z 471.833,A -85,B 0,C 180,E1 -6564.628,E2 -6564.628} C_VEL
LIN {X 0,Y 487.931,Z 475.462,A -85,B 0,C 180,E1 -6565.869,E2 -6565.869} C_VEL
LIN {X 0,Y 487.965,Z 477.339,A -85,B 0,C 180,E1 -6566.696,E2 -6566.696} C_VEL
LIN {X 0,Y 487.933,Z 478.745,A -85,B 0,C 180,E1 -6567.522,E2 -6567.522} C_VEL
LIN {X 0,Y 487.892,Z 479.748,A -85,B 0,C 180,E1 -6568.348,E2 -6568.348} C_VEL
LIN {X 0,Y 487.829,Z 480.581,A -85,B 0,C 180,E1 -6569.998,E2 -6569.998} C_VEL
LIN {X 0,Y 487.892,Z 479.764,A -85,B 0,C 180,E1 -6571.649,E2 -6571.649} C_VEL
LIN {X 0,Y 487.932,Z 478.769,A -85,B 0,C 180,E1 -6572.475,E2 -6572.475} C_VEL
LIN {X 0,Y 487.964,Z 477.37,A -85,B 0,C 180,E1 -6573.301,E2 -6573.301} C_VEL
LIN {X 0,Y 487.919,Z 474.421,A -85,B 0,C 180,E1 -6574.542,E2 -6574.542} C_VEL
LIN {X 0,Y 488.01,Z 470.433,A -85,B 0,C 180,E1 -6575.784,E2 -6575.784} C_VEL
LIN {X 0,Y 488.17,Z 464.298,A -85,B 0,C 180,E1 -6577.235,E2 -6577.235} C_VEL
LIN {X 0,Y 488.342,Z 457.593,A -85,B 0,C 180,E1 -6578.48,E2 -6578.48} C_VEL
LIN {X 0,Y 488.59,Z 449.269,A -85,B 0,C 180,E1 -6579.728,E2 -6579.728} C_VEL
LIN {X 0,Y 488.944,Z 440.736,A -85,B 0,C 180,E1 -6580.767,E2 -6580.767} C_VEL
LIN {X 0,Y 489.4,Z 430.194,A -85,B 0,C 180,E1 -6581.805,E2 -6581.805} C_VEL
LIN {X 0,Y 489.768,Z 418.616,A -85,B 0,C 180,E1 -6582.721,E2 -6582.721} C_VEL
LIN {X 0,Y 490.197,Z 406.361,A -85,B 0,C 180,E1 -6583.47,E2 -6583.47} C_VEL
LIN {X 0,Y 490.588,Z 393.91,A -85,B 0,C 180,E1 -6584.039,E2 -6584.039} C_VEL
LIN {X 0,Y 490.908,Z 381.049,A -85,B 0,C 180,E1 -6584.453,E2 -6584.453} C_VEL
LIN {X 0,Y 491.168,Z 367.385,A -85,B 0,C 180,E1 -6584.71,E2 -6584.71} C_VEL
LIN {X 0,Y 491.546,Z 283.318,A -85,B 0,C 180,E1 -6585.945,E2 -6585.945} C_VEL
LIN {X 0,Y 489.219,Z 267.334,A -85,B 0,C 180,E1 -6586.265,E2 -6586.265} C_VEL
LIN {X 0,Y 489.762,Z 248.389,A -85,B 0,C 180,E1 -6589.268,E2 -6589.268} C_VEL
LIN {X 0,Y 490.384,Z 229.354,A -85,B 0,C 180,E1 -6592.317,E2 -6592.317} C_VEL
LIN {X 0,Y 490.705,Z 219.795,A -85,B 0,C 180,E1 -6593.862,E2 -6593.862} C_VEL
LIN {X 0,Y 489.423,Z 211.86,A -85,B 0,C 180,E1 -6595.221,E2 -6595.221} C_VEL
LIN {X 0,Y 488.792,Z 208.602,A -85,B 0,C 180,E1 -6595.806,E2 -6595.806} C_VEL
LIN {X 0,Y 488.716,Z 208.608,A -85,B 0,C 180,E1 -6598.692,E2 -6598.692} C_VEL
LIN {X 0,Y 488.674,Z 208.609,A -85,B 0,C 180,E1 -6601.176,E2 -6601.176} C_VEL
LIN {X 0,Y 488.714,Z 208.611,A -85,B 0,C 180,E1 -6604.108,E2 -6604.108} C_VEL
LIN {X 0,Y 488.658,Z 208.611,A -85,B 0,C 180,E1 -6607.155,E2 -6607.155} C_VEL
LIN {X 0,Y 488.691,Z 208.61,A -85,B 0,C 180,E1 -6610.341,E2 -6610.341} C_VEL
LIN {X 0,Y 488.655,Z 208.617,A -85,B 0,C 180,E1 -6613.65,E2 -6613.65} C_VEL
LIN {X 0,Y 488.683,Z 208.61,A -85,B 0,C 180,E1 -6616.345,E2 -6616.345} C_VEL
LIN {X 0,Y 488.733,Z 208.609,A -85,B 0,C 180,E1 -6619.676,E2 -6619.676} C_VEL
LIN {X 0,Y 488.643,Z 208.613,A -85,B 0,C 180,E1 -6622.838,E2 -6622.838} C_VEL
LIN {X 0,Y 488.692,Z 208.612,A -85,B 0,C 180,E1 -6625.884,E2 -6625.884} C_VEL
LIN {X 0,Y 488.653,Z 208.612,A -85,B 0,C 180,E1 -6628.817,E2 -6628.817} C_VEL
LIN {X 0,Y 488.7,Z 208.612,A -85,B 0,C 180,E1 -6631.668,E2 -6631.668} C_VEL
LIN {X 0,Y 488.703,Z 208.605,A -85,B 0,C 180,E1 -6634.442,E2 -6634.442} C_VEL
LIN {X 0,Y 488.699,Z 208.61,A -85,B 0,C 180,E1 -6637.152,E2 -6637.152} C_VEL
LIN {X 0,Y 488.697,Z 208.609,A -85,B 0,C 180,E1 -6639.809,E2 -6639.809} C_VEL
LIN {X 0,Y 488.685,Z 208.607,A -85,B 0,C 180,E1 -6642.422,E2 -6642.422} C_VEL
LIN {X 0,Y 488.709,Z 208.609,A -85,B 0,C 180,E1 -6644.998,E2 -6644.998} C_VEL
LIN {X 0,Y 488.779,Z 208.596,A -85,B 0,C 180,E1 -6648.387,E2 -6648.387} C_VEL
LIN {X 0,Y 488.79,Z 208.596,A -85,B 0,C 180,E1 -6651.733,E2 -6651.733} C_VEL
LIN {X 0,Y 488.819,Z 208.591,A -85,B 0,C 180,E1 -6654.224,E2 -6654.224} C_VEL
LIN {X 0,Y 488.906,Z 208.583,A -85,B 0,C 180,E1 -6657.528,E2 -6657.528} C_VEL
LIN {X 0,Y 488.905,Z 208.58,A -85,B 0,C 180,E1 -6660,E2 -6660} C_VEL
LIN {X 0,Y 488.901,Z 208.582,A -85,B 0,C 180,E1 -6662.472,E2 -6662.472} C_VEL
LIN {X 0,Y 488.801,Z 208.593,A -85,B 0,C 180,E1 -6665.776,E2 -6665.776} C_VEL
LIN {X 0,Y 488.759,Z 208.599,A -85,B 0,C 180,E1 -6668.267,E2 -6668.267} C_VEL
LIN {X 0,Y 488.776,Z 208.597,A -85,B 0,C 180,E1 -6671.613,E2 -6671.613} C_VEL
LIN {X 0,Y 488.708,Z 208.61,A -85,B 0,C 180,E1 -6675.002,E2 -6675.002} C_VEL
LIN {X 0,Y 488.701,Z 208.61,A -85,B 0,C 180,E1 -6678.444,E2 -6678.444} C_VEL
LIN {X 0,Y 488.659,Z 208.614,A -85,B 0,C 180,E1 -6681.073,E2 -6681.073} C_VEL
LIN {X 0,Y 488.649,Z 208.612,A -85,B 0,C 180,E1 -6683.748,E2 -6683.748} C_VEL
LIN {X 0,Y 488.75,Z 208.603,A -85,B 0,C 180,E1 -6686.948,E2 -6686.948} C_VEL
LIN {X 0,Y 488.673,Z 208.615,A -85,B 0,C 180,E1 -6690.368,E2 -6690.368} C_VEL
LIN {X 0,Y 488.693,Z 208.606,A -85,B 0,C 180,E1 -6693.488,E2 -6693.488} C_VEL
LIN {X 0,Y 488.648,Z 208.62,A -85,B 0,C 180,E1 -6696.359,E2 -6696.359} C_VEL
LIN {X 0,Y 488.699,Z 208.606,A -85,B 0,C 180,E1 -6699.255,E2 -6699.255} C_VEL
LIN {X 0,Y 488.697,Z 208.611,A -85,B 0,C 180,E1 -6702.525,E2 -6702.525} C_VEL
LIN {X 0,Y 488.68,Z 208.608,A -85,B 0,C 180,E1 -6705.203,E2 -6705.203} C_VEL
LIN {X 0,Y 488.68,Z 208.614,A -85,B 0,C 180,E1 -6708.404,E2 -6708.404} C_VEL
LIN {X 0,Y 488.678,Z 208.609,A -85,B 0,C 180,E1 -6710.952,E2 -6710.952} C_VEL
LIN {X 0,Y 488.662,Z 208.616,A -85,B 0,C 180,E1 -6713.873,E2 -6713.873} C_VEL
LIN {X 0,Y 488.72,Z 208.603,A -85,B 0,C 180,E1 -6716.881,E2 -6716.881} C_VEL
LIN {X 0,Y 488.708,Z 208.61,A -85,B 0,C 180,E1 -6719.785,E2 -6719.785} C_VEL
LIN {X 0,Y 488.779,Z 208.596,A -85,B 0,C 180,E1 -6723.06,E2 -6723.06} C_VEL
LIN {X 0,Y 488.713,Z 208.605,A -85,B 0,C 180,E1 -6724.383,E2 -6724.383} C_VEL
LIN {X 0,Y 488.064,Z 208.69,A -85,B 0,C 180,E1 -6725.071,E2 -6725.071} C_VEL
LIN {X 0,Y 485.201,Z 209.051,A -85,B 0,C 180,E1 -6726.188,E2 -6726.188} C_VEL
LIN {X 0,Y 482.764,Z 209.354,A -85,B 0,C 180,E1 -6727.088,E2 -6727.088} C_VEL
LIN {X 0,Y 481.713,Z 209.484,A -85,B 0,C 180,E1 -6727.784,E2 -6727.784} C_VEL
LIN {X 0,Y 481.626,Z 209.489,A -85,B 0,C 180,E1 -6728.019,E2 -6728.019} C_VEL
LIN {X 0,Y 481.696,Z 209.48,A -85,B 0,C 180,E1 -6730.396,E2 -6730.396} C_VEL
LIN {X 0,Y 481.668,Z 209.482,A -85,B 0,C 180,E1 -6733.036,E2 -6733.036} C_VEL
LIN {X 0,Y 481.68,Z 209.488,A -85,B 0,C 180,E1 -6735.641,E2 -6735.641} C_VEL
LIN {X 0,Y 481.75,Z 209.476,A -85,B 0,C 180,E1 -6738.218,E2 -6738.218} C_VEL
LIN {X 0,Y 481.772,Z 209.541,A -85,B 0,C 180,E1 -6741.403,E2 -6741.403} C_VEL
LIN {X 0,Y 482.556,Z 215.757,A -85,B 0,C 180,E1 -6742.681,E2 -6742.681} C_VEL
LIN {X 0,Y 482.362,Z 225.444,A -85,B 0,C 180,E1 -6744.594,E2 -6744.594} C_VEL
LIN {X 0,Y 484.963,Z 238.896,A -85,B 0,C 180,E1 -6744.884,E2 -6744.884} C_VEL
LIN {X 0,Y 484.203,Z 332.155,A -85,B 0,C 180,E1 -6746.283,E2 -6746.283} C_VEL
LIN {X 0,Y 483.992,Z 345.314,A -85,B 0,C 180,E1 -6746.646,E2 -6746.646} C_VEL
LIN {X 0,Y 483.708,Z 358.471,A -85,B 0,C 180,E1 -6747.191,E2 -6747.191} C_VEL
LIN {X 0,Y 483.395,Z 369.565,A -85,B 0,C 180,E1 -6747.815,E2 -6747.815} C_VEL
LIN {X 0,Y 482.885,Z 381.086,A -85,B 0,C 180,E1 -6748.647,E2 -6748.647} C_VEL
LIN {X 0,Y 482.468,Z 391.435,A -85,B 0,C 180,E1 -6749.584,E2 -6749.584} C_VEL
LIN {X 0,Y 482.099,Z 400.781,A -85,B 0,C 180,E1 -6750.628,E2 -6750.628} C_VEL
LIN {X 0,Y 481.697,Z 409.799,A -85,B 0,C 180,E1 -6751.883,E2 -6751.883} C_VEL
LIN {X 0,Y 481.412,Z 417.075,A -85,B 0,C 180,E1 -6753.14,E2 -6753.14} C_VEL
LIN {X 0,Y 481.209,Z 423.773,A -85,B 0,C 180,E1 -6754.608,E2 -6754.608} C_VEL
LIN {X 0,Y 481.083,Z 428.206,A -85,B 0,C 180,E1 -6755.87,E2 -6755.87} C_VEL
LIN {X 0,Y 481.004,Z 430.552,A -85,B 0,C 180,E1 -6756.714,E2 -6756.714} C_VEL
LIN {X 0,Y 480.918,Z 432.476,A -85,B 0,C 180,E1 -6757.558,E2 -6757.558} C_VEL
LIN {X 0,Y 480.838,Z 433.975,A -85,B 0,C 180,E1 -6758.405,E2 -6758.405} C_VEL
LIN {X 0,Y 480.813,Z 435.02,A -85,B 0,C 180,E1 -6759.253,E2 -6759.253} C_VEL
LIN {X 0,Y 480.819,Z 435.946,A -85,B 0,C 180,E1 -6760.954,E2 -6760.954} C_VEL
LIN {X 0,Y 480.844,Z 435.798,A -85,B 0,C 180,E1 -6761.808,E2 -6761.808} C_VEL
LIN {X 0,Y 480.809,Z 434.243,A -85,B 0,C 180,E1 -6763.525,E2 -6763.525} C_VEL
LIN {X 0,Y 480.891,Z 432.855,A -85,B 0,C 180,E1 -6764.386,E2 -6764.386} C_VEL
LIN {X 0,Y 480.983,Z 430.003,A -85,B 0,C 180,E1 -6765.64,E2 -6765.64} C_VEL
LIN {X 0,Y 481.118,Z 425.826,A -85,B 0,C 180,E1 -6766.987,E2 -6766.987} C_VEL
LIN {X 0,Y 481.368,Z 420.124,A -85,B 0,C 180,E1 -6768.376,E2 -6768.376} C_VEL
LIN {X 0,Y 481.656,Z 412.466,A -85,B 0,C 180,E1 -6769.831,E2 -6769.831} C_VEL
LIN {X 0,Y 482.035,Z 404.187,A -85,B 0,C 180,E1 -6771.074,E2 -6771.074} C_VEL
LIN {X 0,Y 482.508,Z 394.39,A -85,B 0,C 180,E1 -6772.253,E2 -6772.253} C_VEL
LIN {X 0,Y 482.908,Z 384.105,A -85,B 0,C 180,E1 -6773.254,E2 -6773.254} C_VEL
LIN {X 0,Y 483.381,Z 372.623,A -85,B 0,C 180,E1 -6774.136,E2 -6774.136} C_VEL
LIN {X 0,Y 483.758,Z 360.562,A -85,B 0,C 180,E1 -6774.859,E2 -6774.859} C_VEL
LIN {X 0,Y 484.078,Z 348.089,A -85,B 0,C 180,E1 -6775.416,E2 -6775.416} C_VEL
LIN {X 0,Y 484.358,Z 335.204,A -85,B 0,C 180,E1 -6775.803,E2 -6775.803} C_VEL
LIN {X 0,Y 484.563,Z 316.577,A -85,B 0,C 180,E1 -6776.122,E2 -6776.122} C_VEL
LIN {X 0,Y 485.099,Z 238.646,A -85,B 0,C 180,E1 -6777.29,E2 -6777.29} C_VEL
LIN {X 0,Y 482.456,Z 225.427,A -85,B 0,C 180,E1 -6777.614,E2 -6777.614} C_VEL
LIN {X 0,Y 482.477,Z 213.726,A -85,B 0,C 180,E1 -6779.926,E2 -6779.926} C_VEL
LIN {X 0,Y 481.691,Z 209.485,A -85,B 0,C 180,E1 -6780.828,E2 -6780.828} C_VEL
LIN {X 0,Y 481.693,Z 209.482,A -85,B 0,C 180,E1 -6783.732,E2 -6783.732} C_VEL
LIN {X 0,Y 481.623,Z 209.494,A -85,B 0,C 180,E1 -6786.745,E2 -6786.745} C_VEL
LIN {X 0,Y 481.68,Z 209.487,A -85,B 0,C 180,E1 -6789.937,E2 -6789.937} C_VEL
LIN {X 0,Y 481.627,Z 209.489,A -85,B 0,C 180,E1 -6793.298,E2 -6793.298} C_VEL
LIN {X 0,Y 481.67,Z 209.484,A -85,B 0,C 180,E1 -6796.703,E2 -6796.703} C_VEL
LIN {X 0,Y 481.673,Z 209.487,A -85,B 0,C 180,E1 -6800.059,E2 -6800.059} C_VEL
LIN {X 0,Y 481.61,Z 209.489,A -85,B 0,C 180,E1 -6803.251,E2 -6803.251} C_VEL
LIN {X 0,Y 481.69,Z 209.483,A -85,B 0,C 180,E1 -6806.328,E2 -6806.328} C_VEL
LIN {X 0,Y 481.635,Z 209.487,A -85,B 0,C 180,E1 -6809.414,E2 -6809.414} C_VEL
LIN {X 0,Y 481.677,Z 209.482,A -85,B 0,C 180,E1 -6812.166,E2 -6812.166} C_VEL
LIN {X 0,Y 481.693,Z 209.48,A -85,B 0,C 180,E1 -6814.968,E2 -6814.968} C_VEL
LIN {X 0,Y 481.632,Z 209.493,A -85,B 0,C 180,E1 -6817.704,E2 -6817.704} C_VEL
LIN {X 0,Y 481.677,Z 209.478,A -85,B 0,C 180,E1 -6820.392,E2 -6820.392} C_VEL
LIN {X 0,Y 481.668,Z 209.484,A -85,B 0,C 180,E1 -6823.033,E2 -6823.033} C_VEL
LIN {X 0,Y 481.659,Z 209.49,A -85,B 0,C 180,E1 -6825.638,E2 -6825.638} C_VEL
LIN {X 0,Y 481.72,Z 209.474,A -85,B 0,C 180,E1 -6828.214,E2 -6828.214} C_VEL
LIN {X 0,Y 481.732,Z 209.479,A -85,B 0,C 180,E1 -6831.611,E2 -6831.611} C_VEL
LIN {X 0,Y 481.794,Z 209.464,A -85,B 0,C 180,E1 -6834.139,E2 -6834.139} C_VEL
LIN {X 0,Y 481.892,Z 209.455,A -85,B 0,C 180,E1 -6837.492,E2 -6837.492} C_VEL
LIN {X 0,Y 481.871,Z 209.46,A -85,B 0,C 180,E1 -6840.836,E2 -6840.836} C_VEL
LIN {X 0,Y 481.891,Z 209.454,A -85,B 0,C 180,E1 -6842.508,E2 -6842.508} C_VEL
LIN {X 0,Y 481.77,Z 209.469,A -85,B 0,C 180,E1 -6845.861,E2 -6845.861} C_VEL
LIN {X 0,Y 481.707,Z 209.474,A -85,B 0,C 180,E1 -6848.389,E2 -6848.389} C_VEL
LIN {X 0,Y 481.755,Z 209.468,A -85,B 0,C 180,E1 -6851.785,E2 -6851.785} C_VEL
LIN {X 0,Y 481.709,Z 209.479,A -85,B 0,C 180,E1 -6855.225,E2 -6855.225} C_VEL
LIN {X 0,Y 481.677,Z 209.486,A -85,B 0,C 180,E1 -6858.723,E2 -6858.723} C_VEL
LIN {X 0,Y 481.615,Z 209.487,A -85,B 0,C 180,E1 -6861.396,E2 -6861.396} C_VEL
LIN {X 0,Y 481.623,Z 209.49,A -85,B 0,C 180,E1 -6864.116,E2 -6864.116} C_VEL
LIN {X 0,Y 481.668,Z 209.485,A -85,B 0,C 180,E1 -6867.128,E2 -6867.128} C_VEL
LIN {X 0,Y 481.647,Z 209.482,A -85,B 0,C 180,E1 -6869.743,E2 -6869.743} C_VEL
LIN {X 0,Y 481.628,Z 209.49,A -85,B 0,C 180,E1 -6872.678,E2 -6872.678} C_VEL
LIN {X 0,Y 481.614,Z 209.49,A -85,B 0,C 180,E1 -6875.712,E2 -6875.712} C_VEL
LIN {X 0,Y 481.647,Z 209.482,A -85,B 0,C 180,E1 -6878.861,E2 -6878.861} C_VEL
LIN {X 0,Y 481.636,Z 209.49,A -85,B 0,C 180,E1 -6881.914,E2 -6881.914} C_VEL
LIN {X 0,Y 481.64,Z 209.49,A -85,B 0,C 180,E1 -6884.46,E2 -6884.46} C_VEL
LIN {X 0,Y 481.628,Z 209.491,A -85,B 0,C 180,E1 -6887.84,E2 -6887.84} C_VEL
LIN {X 0,Y 481.656,Z 209.483,A -85,B 0,C 180,E1 -6891.142,E2 -6891.142} C_VEL
LIN {X 0,Y 481.63,Z 209.49,A -85,B 0,C 180,E1 -6894.292,E2 -6894.292} C_VEL
LIN {X 0,Y 481.666,Z 209.483,A -85,B 0,C 180,E1 -6897.327,E2 -6897.327} C_VEL
LIN {X 0,Y 481.669,Z 209.488,A -85,B 0,C 180,E1 -6900.26,E2 -6900.26} C_VEL
LIN {X 0,Y 481.688,Z 209.485,A -85,B 0,C 180,E1 -6903.577,E2 -6903.577} C_VEL
LIN {X 0,Y 481.72,Z 209.686,A -85,B 0,C 180,E1 -6903.87,E2 -6903.87} C_VEL
LIN {X 0,Y 483.796,Z 220.154,A -85,B 0,C 180,E1 -6905.772,E2 -6905.772} C_VEL
LIN {X 0,Y 483.716,Z 226.878,A -85,B 0,C 180,E1 -6906.904,E2 -6906.904} C_VEL
LIN {X 0,Y 482.961,Z 245.698,A -85,B 0,C 180,E1 -6910.003,E2 -6910.003} C_VEL
LIN {X 0,Y 482.277,Z 266.323,A -85,B 0,C 180,E1 -6913.35,E2 -6913.35} C_VEL
LIN {X 0,Y 482.257,Z 266.829,A -85,B 0,C 180,E1 -6913.431,E2 -6913.431} C_VEL
LIN {X 0,Y 484.897,Z 285.294,A -85,B 0,C 180,E1 -6913.816,E2 -6913.816} C_VEL
LIN {X 0,Y 484.273,Z 375.347,A -85,B 0,C 180,E1 -6915.18,E2 -6915.18} C_VEL
LIN {X 0,Y 483.926,Z 388.66,A -85,B 0,C 180,E1 -6915.545,E2 -6915.545} C_VEL
LIN {X 0,Y 483.484,Z 401.413,A -85,B 0,C 180,E1 -6916.069,E2 -6916.069} C_VEL
LIN {X 0,Y 483.026,Z 413.876,A -85,B 0,C 180,E1 -6916.773,E2 -6916.773} C_VEL
LIN {X 0,Y 482.569,Z 425.13,A -85,B 0,C 180,E1 -6917.597,E2 -6917.597} C_VEL
LIN {X 0,Y 482.145,Z 435.533,A -85,B 0,C 180,E1 -6918.544,E2 -6918.544} C_VEL
LIN {X 0,Y 481.773,Z 444.068,A -85,B 0,C 180,E1 -6919.493,E2 -6919.493} C_VEL
LIN {X 0,Y 481.382,Z 453.33,A -85,B 0,C 180,E1 -6920.758,E2 -6920.758} C_VEL
LIN {X 0,Y 481.154,Z 460.785,A -85,B 0,C 180,E1 -6922.023,E2 -6922.023} C_VEL
LIN {X 0,Y 480.976,Z 466.777,A -85,B 0,C 180,E1 -6923.286,E2 -6923.286} C_VEL
LIN {X 0,Y 480.925,Z 471.521,A -85,B 0,C 180,E1 -6924.548,E2 -6924.548} C_VEL
LIN {X 0,Y 480.831,Z 475.145,A -85,B 0,C 180,E1 -6925.808,E2 -6925.808} C_VEL
LIN {X 0,Y 480.889,Z 477.019,A -85,B 0,C 180,E1 -6926.647,E2 -6926.647} C_VEL
LIN {X 0,Y 480.845,Z 478.422,A -85,B 0,C 180,E1 -6927.486,E2 -6927.486} C_VEL
LIN {X 0,Y 480.823,Z 479.425,A -85,B 0,C 180,E1 -6928.323,E2 -6928.323} C_VEL
LIN {X 0,Y 480.752,Z 480.255,A -85,B 0,C 180,E1 -6929.998,E2 -6929.998} C_VEL
LIN {X 0,Y 480.823,Z 479.435,A -85,B 0,C 180,E1 -6931.673,E2 -6931.673} C_VEL
LIN {X 0,Y 480.844,Z 478.437,A -85,B 0,C 180,E1 -6932.511,E2 -6932.511} C_VEL
LIN {X 0,Y 480.888,Z 477.036,A -85,B 0,C 180,E1 -6933.349,E2 -6933.349} C_VEL
LIN {X 0,Y 480.837,Z 474.082,A -85,B 0,C 180,E1 -6934.609,E2 -6934.609} C_VEL
LIN {X 0,Y 480.915,Z 470.087,A -85,B 0,C 180,E1 -6935.869,E2 -6935.869} C_VEL
LIN {X 0,Y 481.094,Z 463.94,A -85,B 0,C 180,E1 -6937.342,E2 -6937.342} C_VEL
LIN {X 0,Y 481.285,Z 457.222,A -85,B 0,C 180,E1 -6938.606,E2 -6938.606} C_VEL
LIN {X 0,Y 481.542,Z 448.881,A -85,B 0,C 180,E1 -6939.872,E2 -6939.872} C_VEL
LIN {X 0,Y 481.94,Z 440.326,A -85,B 0,C 180,E1 -6940.925,E2 -6940.925} C_VEL
LIN {X 0,Y 482.401,Z 429.804,A -85,B 0,C 180,E1 -6941.975,E2 -6941.975} C_VEL
LIN {X 0,Y 482.823,Z 417.994,A -85,B 0,C 180,E1 -6942.918,E2 -6942.918} C_VEL
LIN {X 0,Y 483.266,Z 405.815,A -85,B 0,C 180,E1 -6943.666,E2 -6943.666} C_VEL
LIN {X 0,Y 483.698,Z 393.286,A -85,B 0,C 180,E1 -6944.244,E2 -6944.244} C_VEL
LIN {X 0,Y 484.03,Z 380.215,A -85,B 0,C 180,E1 -6944.663,E2 -6944.663} C_VEL
LIN {X 0,Y 484.304,Z 364.41,A -85,B 0,C 180,E1 -6944.95,E2 -6944.95} C_VEL
LIN {X 0,Y 484.593,Z 283.394,A -85,B 0,C 180,E1 -6946.159,E2 -6946.159} C_VEL
LIN {X 0,Y 482.209,Z 266.907,A -85,B 0,C 180,E1 -6946.508,E2 -6946.508} C_VEL
LIN {X 0,Y 482.759,Z 249.269,A -85,B 0,C 180,E1 -6949.344,E2 -6949.344} C_VEL
LIN {X 0,Y 483.366,Z 231.615,A -85,B 0,C 180,E1 -6952.208,E2 -6952.208} C_VEL
LIN {X 0,Y 483.726,Z 220.681,A -85,B 0,C 180,E1 -6954,E2 -6954} C_VEL
LIN {X 0,Y 481.737,Z 209.481,A -85,B 0,C 180,E1 -6955.98,E2 -6955.98} C_VEL
LIN {X 0,Y 481.662,Z 209.486,A -85,B 0,C 180,E1 -6958.899,E2 -6958.899} C_VEL
LIN {X 0,Y 481.638,Z 209.492,A -85,B 0,C 180,E1 -6962.185,E2 -6962.185} C_VEL
LIN {X 0,Y 481.672,Z 209.482,A -85,B 0,C 180,E1 -6964.678,E2 -6964.678} C_VEL
LIN {X 0,Y 481.631,Z 209.494,A -85,B 0,C 180,E1 -6968.003,E2 -6968.003} C_VEL
LIN {X 0,Y 481.629,Z 209.487,A -85,B 0,C 180,E1 -6971.038,E2 -6971.038} C_VEL
LIN {X 0,Y 481.628,Z 209.488,A -85,B 0,C 180,E1 -6974.453,E2 -6974.453} C_VEL
LIN {X 0,Y 481.655,Z 209.483,A -85,B 0,C 180,E1 -6976.842,E2 -6976.842} C_VEL
LIN {X 0,Y 481.676,Z 209.485,A -85,B 0,C 180,E1 -6980.059,E2 -6980.059} C_VEL
LIN {X 0,Y 481.591,Z 209.495,A -85,B 0,C 180,E1 -6983.372,E2 -6983.372} C_VEL
LIN {X 0,Y 481.667,Z 209.482,A -85,B 0,C 180,E1 -6986.327,E2 -6986.327} C_VEL
LIN {X 0,Y 481.614,Z 209.494,A -85,B 0,C 180,E1 -6989.412,E2 -6989.412} C_VEL
LIN {X 0,Y 481.655,Z 209.484,A -85,B 0,C 180,E1 -6992.165,E2 -6992.165} C_VEL
LIN {X 0,Y 481.673,Z 209.483,A -85,B 0,C 180,E1 -6994.967,E2 -6994.967} C_VEL
LIN {X 0,Y 481.627,Z 209.491,A -85,B 0,C 180,E1 -6997.704,E2 -6997.704} C_VEL
LIN {X 0,Y 481.664,Z 209.482,A -85,B 0,C 180,E1 -7000.391,E2 -7000.391} C_VEL
LIN {X 0,Y 481.643,Z 209.489,A -85,B 0,C 180,E1 -7003.032,E2 -7003.032} C_VEL
LIN {X 0,Y 481.641,Z 209.489,A -85,B 0,C 180,E1 -7005.637,E2 -7005.637} C_VEL
LIN {X 0,Y 481.741,Z 209.472,A -85,B 0,C 180,E1 -7008.215,E2 -7008.215} C_VEL
LIN {X 0,Y 481.732,Z 209.477,A -85,B 0,C 180,E1 -7011.611,E2 -7011.611} C_VEL
LIN {X 0,Y 481.778,Z 209.468,A -85,B 0,C 180,E1 -7014.139,E2 -7014.139} C_VEL
LIN {X 0,Y 481.874,Z 209.459,A -85,B 0,C 180,E1 -7017.492,E2 -7017.492} C_VEL
LIN {X 0,Y 481.877,Z 209.456,A -85,B 0,C 180,E1 -7020,E2 -7020} C_VEL
LIN {X 0,Y 481.868,Z 209.459,A -85,B 0,C 180,E1 -7022.508,E2 -7022.508} C_VEL
LIN {X 0,Y 481.761,Z 209.47,A -85,B 0,C 180,E1 -7025.861,E2 -7025.861} C_VEL
LIN {X 0,Y 481.705,Z 209.479,A -85,B 0,C 180,E1 -7028.389,E2 -7028.389} C_VEL
LIN {X 0,Y 481.74,Z 209.473,A -85,B 0,C 180,E1 -7031.785,E2 -7031.785} C_VEL
LIN {X 0,Y 481.688,Z 209.482,A -85,B 0,C 180,E1 -7035.226,E2 -7035.226} C_VEL
LIN {X 0,Y 481.658,Z 209.491,A -85,B 0,C 180,E1 -7038.724,E2 -7038.724} C_VEL
LIN {X 0,Y 481.601,Z 209.491,A -85,B 0,C 180,E1 -7041.397,E2 -7041.397} C_VEL
LIN {X 0,Y 481.63,Z 209.488,A -85,B 0,C 180,E1 -7044.116,E2 -7044.116} C_VEL
LIN {X 0,Y 481.704,Z 209.479,A -85,B 0,C 180,E1 -7047.143,E2 -7047.143} C_VEL
LIN {X 0,Y 481.642,Z 209.485,A -85,B 0,C 180,E1 -7049.744,E2 -7049.744} C_VEL
LIN {X 0,Y 481.629,Z 209.492,A -85,B 0,C 180,E1 -7052.678,E2 -7052.678} C_VEL
LIN {X 0,Y 481.602,Z 209.491,A -85,B 0,C 180,E1 -7055.713,E2 -7055.713} C_VEL
LIN {X 0,Y 481.673,Z 209.481,A -85,B 0,C 180,E1 -7059.357,E2 -7059.357} C_VEL
LIN {X 0,Y 481.639,Z 209.492,A -85,B 0,C 180,E1 -7062.162,E2 -7062.162} C_VEL
LIN {X 0,Y 481.628,Z 209.492,A -85,B 0,C 180,E1 -7064.461,E2 -7064.461} C_VEL
LIN {X 0,Y 481.619,Z 209.491,A -85,B 0,C 180,E1 -7067.843,E2 -7067.843} C_VEL
LIN {X 0,Y 481.654,Z 209.485,A -85,B 0,C 180,E1 -7070.655,E2 -7070.655} C_VEL
LIN {X 0,Y 481.608,Z 209.49,A -85,B 0,C 180,E1 -7073.38,E2 -7073.38} C_VEL
LIN {X 0,Y 481.691,Z 209.483,A -85,B 0,C 180,E1 -7076.334,E2 -7076.334} C_VEL
LIN {X 0,Y 481.634,Z 209.487,A -85,B 0,C 180,E1 -7079.422,E2 -7079.422} C_VEL
LIN {X 0,Y 481.686,Z 209.485,A -85,B 0,C 180,E1 -7082.172,E2 -7082.172} C_VEL
LIN {X 0,Y 481.682,Z 209.48,A -85,B 0,C 180,E1 -7084.972,E2 -7084.972} C_VEL
LIN {X 0,Y 481.626,Z 209.489,A -85,B 0,C 180,E1 -7088.019,E2 -7088.019} C_VEL
LIN {X 0,Y 480.961,Z 209.571,A -85,B 0,C 180,E1 -7088.717,E2 -7088.717} C_VEL
LIN {X 0,Y 478.135,Z 209.93,A -85,B 0,C 180,E1 -7089.851,E2 -7089.851} C_VEL
LIN {X 0,Y 475.747,Z 210.224,A -85,B 0,C 180,E1 -7090.766,E2 -7090.766} C_VEL
LIN {X 0,Y 474.722,Z 210.351,A -85,B 0,C 180,E1 -7091.471,E2 -7091.471} C_VEL
LIN {X 0,Y 474.638,Z 210.362,A -85,B 0,C 180,E1 -7091.71,E2 -7091.71} C_VEL
LIN {X 0,Y 474.695,Z 210.351,A -85,B 0,C 180,E1 -7094.547,E2 -7094.547} C_VEL
LIN {X 0,Y 474.703,Z 210.356,A -85,B 0,C 180,E1 -7098.04,E2 -7098.04} C_VEL
LIN {X 0,Y 474.751,Z 210.45,A -85,B 0,C 180,E1 -7101.275,E2 -7101.275} C_VEL
LIN {X 0,Y 475.566,Z 216.709,A -85,B 0,C 180,E1 -7102.573,E2 -7102.573} C_VEL
LIN {X 0,Y 475.376,Z 225.777,A -85,B 0,C 180,E1 -7104.368,E2 -7104.368} C_VEL
LIN {X 0,Y 478.135,Z 240.034,A -85,B 0,C 180,E1 -7104.678,E2 -7104.678} C_VEL
LIN {X 0,Y 477.303,Z 333.057,A -85,B 0,C 180,E1 -7106.097,E2 -7106.097} C_VEL
LIN {X 0,Y 477.09,Z 346.018,A -85,B 0,C 180,E1 -7106.465,E2 -7106.465} C_VEL
LIN {X 0,Y 476.806,Z 358.527,A -85,B 0,C 180,E1 -7106.992,E2 -7106.992} C_VEL
LIN {X 0,Y 476.441,Z 370.49,A -85,B 0,C 180,E1 -7107.677,E2 -7107.677} C_VEL
LIN {X 0,Y 475.919,Z 381.902,A -85,B 0,C 180,E1 -7108.521,E2 -7108.521} C_VEL
LIN {X 0,Y 475.478,Z 392.173,A -85,B 0,C 180,E1 -7109.472,E2 -7109.472} C_VEL
LIN {X 0,Y 475.11,Z 400.585,A -85,B 0,C 180,E1 -7110.425,E2 -7110.425} C_VEL
LIN {X 0,Y 474.744,Z 408.361,A -85,B 0,C 180,E1 -7111.486,E2 -7111.486} C_VEL
LIN {X 0,Y 474.392,Z 415.974,A -85,B 0,C 180,E1 -7112.761,E2 -7112.761} C_VEL
LIN {X 0,Y 474.207,Z 422.979,A -85,B 0,C 180,E1 -7114.251,E2 -7114.251} C_VEL
LIN {X 0,Y 473.998,Z 427.669,A -85,B 0,C 180,E1 -7115.532,E2 -7115.532} C_VEL
LIN {X 0,Y 473.904,Z 431.257,A -85,B 0,C 180,E1 -7116.815,E2 -7116.815} C_VEL
LIN {X 0,Y 473.828,Z 433.113,A -85,B 0,C 180,E1 -7117.672,E2 -7117.672} C_VEL
LIN {X 0,Y 473.752,Z 434.502,A -85,B 0,C 180,E1 -7118.532,E2 -7118.532} C_VEL
LIN {X 0,Y 473.712,Z 436.091,A -85,B 0,C 180,E1 -7120.256,E2 -7120.256} C_VEL
LIN {X 0,Y 473.765,Z 436.165,A -85,B 0,C 180,E1 -7121.742,E2 -7121.742} C_VEL
LIN {X 0,Y 473.707,Z 435.404,A -85,B 0,C 180,E1 -7122.859,E2 -7122.859} C_VEL
LIN {X 0,Y 473.733,Z 434.368,A -85,B 0,C 180,E1 -7123.731,E2 -7123.731} C_VEL
LIN {X 0,Y 473.827,Z 432.873,A -85,B 0,C 180,E1 -7124.605,E2 -7124.605} C_VEL
LIN {X 0,Y 473.94,Z 429.788,A -85,B 0,C 180,E1 -7125.922,E2 -7125.922} C_VEL
LIN {X 0,Y 474.08,Z 425.577,A -85,B 0,C 180,E1 -7127.247,E2 -7127.247} C_VEL
LIN {X 0,Y 474.377,Z 419.488,A -85,B 0,C 180,E1 -7128.707,E2 -7128.707} C_VEL
LIN {X 0,Y 474.641,Z 413.174,A -85,B 0,C 180,E1 -7129.911,E2 -7129.911} C_VEL
LIN {X 0,Y 475.045,Z 405.317,A -85,B 0,C 180,E1 -7131.13,E2 -7131.13} C_VEL
LIN {X 0,Y 475.454,Z 396.343,A -85,B 0,C 180,E1 -7132.258,E2 -7132.258} C_VEL
LIN {X 0,Y 475.901,Z 386.448,A -85,B 0,C 180,E1 -7133.268,E2 -7133.268} C_VEL
LIN {X 0,Y 476.454,Z 374.954,A -85,B 0,C 180,E1 -7134.208,E2 -7134.208} C_VEL
LIN {X 0,Y 476.849,Z 363.234,A -85,B 0,C 180,E1 -7134.953,E2 -7134.953} C_VEL
LIN {X 0,Y 477.202,Z 350.48,A -85,B 0,C 180,E1 -7135.563,E2 -7135.563} C_VEL
LIN {X 0,Y 477.528,Z 337.27,A -85,B 0,C 180,E1 -7135.997,E2 -7135.997} C_VEL
LIN {X 0,Y 477.687,Z 322.429,A -85,B 0,C 180,E1 -7136.279,E2 -7136.279} C_VEL
LIN {X 0,Y 478.321,Z 239.172,A -85,B 0,C 180,E1 -7137.546,E2 -7137.546} C_VEL
LIN {X 0,Y 475.518,Z 225.801,A -85,B 0,C 180,E1 -7137.873,E2 -7137.873} C_VEL
LIN {X 0,Y 475.59,Z 215.513,A -85,B 0,C 180,E1 -7139.922,E2 -7139.922} C_VEL
LIN {X 0,Y 474.666,Z 210.359,A -85,B 0,C 180,E1 -7141.035,E2 -7141.035} C_VEL
LIN {X 0,Y 474.629,Z 210.365,A -85,B 0,C 180,E1 -7144.239,E2 -7144.239} C_VEL
LIN {X 0,Y 474.586,Z 210.368,A -85,B 0,C 180,E1 -7147.382,E2 -7147.382} C_VEL
LIN {X 0,Y 474.642,Z 210.363,A -85,B 0,C 180,E1 -7149.649,E2 -7149.649} C_VEL
LIN {X 0,Y 474.604,Z 210.365,A -85,B 0,C 180,E1 -7152.932,E2 -7152.932} C_VEL
LIN {X 0,Y 474.605,Z 210.368,A -85,B 0,C 180,E1 -7155.894,E2 -7155.894} C_VEL
LIN {X 0,Y 474.63,Z 210.36,A -85,B 0,C 180,E1 -7159.036,E2 -7159.036} C_VEL
LIN {X 0,Y 474.599,Z 210.368,A -85,B 0,C 180,E1 -7161.701,E2 -7161.701} C_VEL
LIN {X 0,Y 474.61,Z 210.362,A -85,B 0,C 180,E1 -7164.724,E2 -7164.724} C_VEL
LIN {X 0,Y 474.616,Z 210.368,A -85,B 0,C 180,E1 -7167.786,E2 -7167.786} C_VEL
LIN {X 0,Y 474.608,Z 210.362,A -85,B 0,C 180,E1 -7170.881,E2 -7170.881} C_VEL
LIN {X 0,Y 474.636,Z 210.362,A -85,B 0,C 180,E1 -7173.627,E2 -7173.627} C_VEL
LIN {X 0,Y 474.61,Z 210.358,A -85,B 0,C 180,E1 -7176.64,E2 -7176.64} C_VEL
LIN {X 0,Y 474.626,Z 210.358,A -85,B 0,C 180,E1 -7180.088,E2 -7180.088} C_VEL
LIN {X 0,Y 474.626,Z 210.36,A -85,B 0,C 180,E1 -7182.773,E2 -7182.773} C_VEL
LIN {X 0,Y 474.617,Z 210.363,A -85,B 0,C 180,E1 -7185.42,E2 -7185.42} C_VEL
LIN {X 0,Y 474.673,Z 210.353,A -85,B 0,C 180,E1 -7188.037,E2 -7188.037} C_VEL
LIN {X 0,Y 474.697,Z 210.357,A -85,B 0,C 180,E1 -7191.486,E2 -7191.486} C_VEL
LIN {X 0,Y 474.758,Z 210.341,A -85,B 0,C 180,E1 -7194.052,E2 -7194.052} C_VEL
LIN {X 0,Y 474.859,Z 210.332,A -85,B 0,C 180,E1 -7197.455,E2 -7197.455} C_VEL
LIN {X 0,Y 474.823,Z 210.338,A -85,B 0,C 180,E1 -7200.848,E2 -7200.848} C_VEL
LIN {X 0,Y 474.857,Z 210.33,A -85,B 0,C 180,E1 -7202.545,E2 -7202.545} C_VEL
LIN {X 0,Y 474.732,Z 210.346,A -85,B 0,C 180,E1 -7205.948,E2 -7205.948} C_VEL
LIN {X 0,Y 474.679,Z 210.351,A -85,B 0,C 180,E1 -7208.514,E2 -7208.514} C_VEL
LIN {X 0,Y 474.699,Z 210.347,A -85,B 0,C 180,E1 -7211.963,E2 -7211.963} C_VEL
LIN {X 0,Y 474.649,Z 210.355,A -85,B 0,C 180,E1 -7215.768,E2 -7215.768} C_VEL
LIN {X 0,Y 474.632,Z 210.364,A -85,B 0,C 180,E1 -7219.012,E2 -7219.012} C_VEL
LIN {X 0,Y 474.558,Z 210.365,A -85,B 0,C 180,E1 -7221.73,E2 -7221.73} C_VEL
LIN {X 0,Y 474.602,Z 210.368,A -85,B 0,C 180,E1 -7224.496,E2 -7224.496} C_VEL
LIN {X 0,Y 474.612,Z 210.362,A -85,B 0,C 180,E1 -7227.325,E2 -7227.325} C_VEL
LIN {X 0,Y 474.576,Z 210.366,A -85,B 0,C 180,E1 -7230.232,E2 -7230.232} C_VEL
LIN {X 0,Y 474.592,Z 210.361,A -85,B 0,C 180,E1 -7233.224,E2 -7233.224} C_VEL
LIN {X 0,Y 474.567,Z 210.372,A -85,B 0,C 180,E1 -7236.326,E2 -7236.326} C_VEL
LIN {X 0,Y 474.592,Z 210.359,A -85,B 0,C 180,E1 -7239.647,E2 -7239.647} C_VEL
LIN {X 0,Y 474.608,Z 210.368,A -85,B 0,C 180,E1 -7242.238,E2 -7242.238} C_VEL
LIN {X 0,Y 474.602,Z 210.361,A -85,B 0,C 180,E1 -7245.3,E2 -7245.3} C_VEL
LIN {X 0,Y 474.597,Z 210.365,A -85,B 0,C 180,E1 -7248.215,E2 -7248.215} C_VEL
LIN {X 0,Y 474.6,Z 210.364,A -85,B 0,C 180,E1 -7251.544,E2 -7251.544} C_VEL
LIN {X 0,Y 474.618,Z 210.362,A -85,B 0,C 180,E1 -7254.727,E2 -7254.727} C_VEL
LIN {X 0,Y 474.63,Z 210.364,A -85,B 0,C 180,E1 -7257.789,E2 -7257.789} C_VEL
LIN {X 0,Y 474.603,Z 210.365,A -85,B 0,C 180,E1 -7260.89,E2 -7260.89} C_VEL
LIN {X 0,Y 474.692,Z 210.554,A -85,B 0,C 180,E1 -7263.631,E2 -7263.631} C_VEL
LIN {X 0,Y 476.836,Z 221.342,A -85,B 0,C 180,E1 -7265.627,E2 -7265.627} C_VEL
LIN {X 0,Y 476.858,Z 226.717,A -85,B 0,C 180,E1 -7266.552,E2 -7266.552} C_VEL
LIN {X 0,Y 476.065,Z 244.169,A -85,B 0,C 180,E1 -7269.476,E2 -7269.476} C_VEL
LIN {X 0,Y 475.462,Z 261.619,A -85,B 0,C 180,E1 -7272.361,E2 -7272.361} C_VEL
LIN {X 0,Y 475.294,Z 266.481,A -85,B 0,C 180,E1 -7273.158,E2 -7273.158} C_VEL
LIN {X 0,Y 478.116,Z 286.235,A -85,B 0,C 180,E1 -7273.579,E2 -7273.579} C_VEL
LIN {X 0,Y 477.439,Z 375.764,A -85,B 0,C 180,E1 -7274.963,E2 -7274.963} C_VEL
LIN {X 0,Y 477.051,Z 389.577,A -85,B 0,C 180,E1 -7275.36,E2 -7275.36} C_VEL
LIN {X 0,Y 476.593,Z 401.434,A -85,B 0,C 180,E1 -7275.863,E2 -7275.863} C_VEL
LIN {X 0,Y 476.119,Z 413.468,A -85,B 0,C 180,E1 -7276.556,E2 -7276.556} C_VEL
LIN {X 0,Y 475.655,Z 424.395,A -85,B 0,C 180,E1 -7277.364,E2 -7277.364} C_VEL
LIN {X 0,Y 475.169,Z 435.346,A -85,B 0,C 180,E1 -7278.374,E2 -7278.374} C_VEL
LIN {X 0,Y 474.746,Z 443.849,A -85,B 0,C 180,E1 -7279.336,E2 -7279.336} C_VEL
LIN {X 0,Y 474.345,Z 453.079,A -85,B 0,C 180,E1 -7280.619,E2 -7280.619} C_VEL
LIN {X 0,Y 474.085,Z 460.516,A -85,B 0,C 180,E1 -7281.903,E2 -7281.903} C_VEL
LIN {X 0,Y 473.901,Z 466.494,A -85,B 0,C 180,E1 -7283.185,E2 -7283.185} C_VEL
LIN {X 0,Y 473.838,Z 471.225,A -85,B 0,C 180,E1 -7284.467,E2 -7284.467} C_VEL
LIN {X 0,Y 473.736,Z 474.84,A -85,B 0,C 180,E1 -7285.745,E2 -7285.745} C_VEL
LIN {X 0,Y 473.796,Z 476.708,A -85,B 0,C 180,E1 -7286.597,E2 -7286.597} C_VEL
LIN {X 0,Y 473.756,Z 479.107,A -85,B 0,C 180,E1 -7288.298,E2 -7288.298} C_VEL
LIN {X 0,Y 473.678,Z 479.929,A -85,B 0,C 180,E1 -7289.998,E2 -7289.998} C_VEL
LIN {X 0,Y 473.756,Z 479.101,A -85,B 0,C 180,E1 -7291.698,E2 -7291.698} C_VEL
LIN {X 0,Y 473.76,Z 478.099,A -85,B 0,C 180,E1 -7292.549,E2 -7292.549} C_VEL
LIN {X 0,Y 473.795,Z 476.691,A -85,B 0,C 180,E1 -7293.4,E2 -7293.4} C_VEL
LIN {X 0,Y 473.76,Z 473.73,A -85,B 0,C 180,E1 -7294.678,E2 -7294.678} C_VEL
LIN {X 0,Y 473.822,Z 469.725,A -85,B 0,C 180,E1 -7295.957,E2 -7295.957} C_VEL
LIN {X 0,Y 473.999,Z 463.559,A -85,B 0,C 180,E1 -7297.452,E2 -7297.452} C_VEL
LIN {X 0,Y 474.196,Z 456.823,A -85,B 0,C 180,E1 -7298.735,E2 -7298.735} C_VEL
LIN {X 0,Y 474.482,Z 448.462,A -85,B 0,C 180,E1 -7300.02,E2 -7300.02} C_VEL
LIN {X 0,Y 474.926,Z 439.875,A -85,B 0,C 180,E1 -7301.089,E2 -7301.089} C_VEL
LIN {X 0,Y 475.389,Z 429.556,A -85,B 0,C 180,E1 -7302.132,E2 -7302.132} C_VEL
LIN {X 0,Y 475.802,Z 418.754,A -85,B 0,C 180,E1 -7303.015,E2 -7303.015} C_VEL
LIN {X 0,Y 476.273,Z 407.186,A -85,B 0,C 180,E1 -7303.762,E2 -7303.762} C_VEL
LIN {X 0,Y 476.694,Z 395.178,A -85,B 0,C 180,E1 -7304.348,E2 -7304.348} C_VEL
LIN {X 0,Y 477.056,Z 382.183,A -85,B 0,C 180,E1 -7304.801,E2 -7304.801} C_VEL
LIN {X 0,Y 477.382,Z 370.038,A -85,B 0,C 180,E1 -7305.063,E2 -7305.063} C_VEL
LIN {X 0,Y 477.798,Z 284.612,A -85,B 0,C 180,E1 -7306.355,E2 -7306.355} C_VEL
LIN {X 0,Y 475.221,Z 266.613,A -85,B 0,C 180,E1 -7306.733,E2 -7306.733} C_VEL
LIN {X 0,Y 475.847,Z 247.482,A -85,B 0,C 180,E1 -7309.855,E2 -7309.855} C_VEL
LIN {X 0,Y 476.462,Z 229.762,A -85,B 0,C 180,E1 -7312.776,E2 -7312.776} C_VEL
LIN {X 0,Y 476.754,Z 221.795,A -85,B 0,C 180,E1 -7314.102,E2 -7314.102} C_VEL
LIN {X 0,Y 474.695,Z 210.357,A -85,B 0,C 180,E1 -7316.145,E2 -7316.145} C_VEL
LIN {X 0,Y 474.608,Z 210.364,A -85,B 0,C 180,E1 -7319.111,E2 -7319.111} C_VEL
LIN {X 0,Y 474.596,Z 210.366,A -85,B 0,C 180,E1 -7322.427,E2 -7322.427} C_VEL
LIN {X 0,Y 474.598,Z 210.364,A -85,B 0,C 180,E1 -7325.466,E2 -7325.466} C_VEL
LIN {X 0,Y 474.587,Z 210.366,A -85,B 0,C 180,E1 -7328.453,E2 -7328.453} C_VEL
LIN {X 0,Y 474.6,Z 210.362,A -85,B 0,C 180,E1 -7330.955,E2 -7330.955} C_VEL
LIN {X 0,Y 474.578,Z 210.37,A -85,B 0,C 180,E1 -7334.101,E2 -7334.101} C_VEL
LIN {X 0,Y 474.618,Z 210.36,A -85,B 0,C 180,E1 -7337.066,E2 -7337.066} C_VEL
LIN {X 0,Y 474.645,Z 210.357,A -85,B 0,C 180,E1 -7340.454,E2 -7340.454} C_VEL
LIN {X 0,Y 474.552,Z 210.377,A -85,B 0,C 180,E1 -7343.673,E2 -7343.673} C_VEL
LIN {X 0,Y 474.601,Z 210.362,A -85,B 0,C 180,E1 -7346.777,E2 -7346.777} C_VEL
LIN {X 0,Y 474.569,Z 210.372,A -85,B 0,C 180,E1 -7349.767,E2 -7349.767} C_VEL
LIN {X 0,Y 474.65,Z 210.356,A -85,B 0,C 180,E1 -7352.677,E2 -7352.677} C_VEL
LIN {X 0,Y 474.618,Z 210.368,A -85,B 0,C 180,E1 -7355.505,E2 -7355.505} C_VEL
LIN {X 0,Y 474.643,Z 210.362,A -85,B 0,C 180,E1 -7359.184,E2 -7359.184} C_VEL
LIN {X 0,Y 474.605,Z 210.363,A -85,B 0,C 180,E1 -7361.882,E2 -7361.882} C_VEL
LIN {X 0,Y 474.645,Z 210.357,A -85,B 0,C 180,E1 -7364.543,E2 -7364.543} C_VEL
